GLOBALCONSTANTS Manufacturer_IDs (* ISOBUS Manufacturer ID defines *)
  (* Standard: 61499-1 *)
  (* Version 1.0, 2026-06-29, Franz Höpfinger, Demmler Andreas Fahrzeugbau *)
  PACKAGE isobus::pgn::const;
  VAR_GLOBAL CONSTANT
    M_FOR_EXPERIMENTAL_OR_DEVELOPMENTAL_USE_ONLY : UINT := 0; (* Manufacturer: For experimental or developmental use only. - 2025-11-06 *)
    M_BENDIX_COMMERCIAL_VEHICLE_SYSTEMS : UINT := 1; (* Manufacturer: Bendix Commercial Vehicle Systems LLC (formerly Allied Signal Inc.) | Location: *)
    M_ALLISON_TRANSMISSION : UINT := 2; (* Manufacturer: Allison Transmission, Inc. | Location: Indianapolis, IN USA - 2015-04-28 *)
    M_AMETEK_US_GAUGE_DIVISION : UINT := 3; (* Manufacturer: Ametek, US Gauge Division | Location: Sellersville, PA USA *)
    M_AMETEK_DIXSON : UINT := 4; (* Manufacturer: Ametek-Dixson | Location: Grand Junction, CO USA *)
    M_AMP : UINT := 5; (* Manufacturer: AMP Inc. | Location: Harrisburg, PA USA *)
    M_BERIFORS_ELECTRONICS : UINT := 6; (* Manufacturer: Berifors Electronics AB | Location: Stockholm, Sweden *)
    M_CASE : UINT := 7; (* Manufacturer: Case Corp. | Location: Burr Ridge, IL USA *)
    M_CATERPILLAR : UINT := 8; (* Manufacturer: Caterpillar Inc. | Location: Peoria, IL USA *)
    M_CHRYSLER : UINT := 9; (* Manufacturer: Chrysler Corp. | Location: Auburn Hills, MI USA *)
    M_CUMMINS : UINT := 10; (* Manufacturer: Cummins Inc (formerly Cummins Engine Co) | Location: Columbus, IN USA *)
    M_DEARBORN_GROUP : UINT := 11; (* Manufacturer: Dearborn Group Inc. | Location: Indianapolis, IN & Farmington Hills, MI USA *)
    M_DEERE_AND_COMPANY_PRECISION_FARMING : UINT := 12; (* Manufacturer: Deere & Company, Precision Farming | Location: East Moline, IL USA *)
    M_DELCO_ELECTRONICS : UINT := 13; (* Manufacturer: Delco Electronics | Location: Kokomo, IN USA *)
    M_DETROIT_DIESEL : UINT := 14; (* Manufacturer: Detroit Diesel Corporation | Location: Detroit, MI USA *)
    M_DICKEY_JOHN : UINT := 15; (* Manufacturer: DICKEY-john Corporation | Location: Auburn, IL USA - 2015-07-27 *)
    M_EATON : UINT := 16; (* Manufacturer: Eaton Corp | Location: Southfield, MI USA *)
    M_EATON_RES_AND_DEV : UINT := 17; (* Manufacturer: Eaton Corp, Corp Res & Dev | Location: Milwaukee, WI USA *)
    M_EATON_TRANSMISSION_DIV : UINT := 18; (* Manufacturer: Eaton Corp, Transmission Div. | Location: Kalamazoo, MI USA *)
    M_EATON_TRUCKING_INFO_SERVICES : UINT := 19; (* Manufacturer: Eaton Corp. Trucking Info Services | Location: Clemmons, NC USA *)
    M_EATON_20 : UINT := 20; (* Manufacturer: Eaton Ltd | Location: Worsley, England *)
    M_ECHLIN_MIDLAND_BRAKE : UINT := 21; (* Manufacturer: Echlin Inc., Midland Brake Inc. | Location: Kansas City, MO USA *)
    M_FORD_MOTOR_ELECTRONIC_CONCEPTS_AND_SYSTEMS : UINT := 22; (* Manufacturer: Ford Motor Co., Electronic Concepts & Systems | Location: Dearborn, MI USA *)
    M_FORD_MOTOR_HEAVY_TRUCK : UINT := 23; (* Manufacturer: Ford Motor Co., Heavy Truck | Location: Dearborn, MI USA *)
    M_FORD_MOTOR_VEHICLE_CONTROLS : UINT := 24; (* Manufacturer: Ford Motor Co., Vehicle Controls | Location: Dearborn, MI USA *)
    M_DAIMLER_TRUCKS_NORTH_AMERICA : UINT := 25; (* Manufacturer: Daimler Trucks North America LLC (formerly Freightliner LLC) | Location: Portland, *)
    M_GENERAL_MOTORS_SERVICE_TECHNOLOGY_GRP : UINT := 26; (* Manufacturer: General Motors Corp, Service Technology Grp | Location: Romulus, MI USA *)
    M_GMC : UINT := 27; (* Manufacturer: GMC | Location: Troy, MI USA *)
    M_GROTE_IND : UINT := 28; (* Manufacturer: Grote Ind. Inc. | Location: Madison, IN USA *)
    M_HINO_MOTORS : UINT := 29; (* Manufacturer: Hino Motors Ltd. | Location: Tokyo, Japan *)
    M_ISUZU_MOTORS : UINT := 30; (* Manufacturer: Isuzu Motors Ltd | Location: Kawasaki, Japan *)
    M_J_POLLAK : UINT := 31; (* Manufacturer: J Pollak Corp | Location: Boston, MA USA *)
    M_JACOBS_VEHICLE_SYSTEMS : UINT := 32; (* Manufacturer: Jacobs Vehicle Systems | Location: Bloomfield, CT USA - 1998-07-01 *)
    M_JOHN_DEERE : UINT := 33; (* Manufacturer: John Deere | Location: Moline, IL USA - 2015-06-29 *)
    M_KELSEY_HAYES : UINT := 34; (* Manufacturer: Kelsey Hayes Co. | Location: Livonia, MI USA *)
    M_KENWORTH_TRUCK : UINT := 35; (* Manufacturer: Kenworth Truck Co. | Location: Kirkland, WA USA *)
    M_LUCAS_IND : UINT := 36; (* Manufacturer: Lucas Ind. | Location: Solihull, W Midlands UK *)
    M_MACK_TRUCKS : UINT := 37; (* Manufacturer: Mack Trucks Inc. | Location: Hagerstown, MD USA *)
    M_MICRO_PROCESSOR_SYSTEMS : UINT := 38; (* Manufacturer: Micro Processor Systems Inc. | Location: Sterling Hts, MI USA *)
    M_MICROFIRM : UINT := 39; (* Manufacturer: Microfirm Inc. | Location: Stillwater, OK USA *)
    M_MOTOROLA_AIEG : UINT := 40; (* Manufacturer: Motorola AIEG Inc. | Location: Northbrook, IL USA *)
    M_MOTOROLA : UINT := 41; (* Manufacturer: Motorola Inc. | Location: Schaumburg, IL USA *)
    M_INTERNATIONAL_TRUCK_AND_ENGINE_ENGINE_ELECTRONICS : UINT := 42; (* Manufacturer: International Truck and Engine Corporation - Engine Electronics (formerly Navistar *)
    M_INTERNATIONAL_TRUCK_AND_ENGINE_VEHICLE_ELECTRONICS : UINT := 43; (* Manufacturer: International Truck and Engine Corporation - Vehicle Electronics (formerly Navistar *)
    M_NIPPONDENSO : UINT := 44; (* Manufacturer: Nippondenso Co. Ltd. | Location: Kariya, Aichi Japan *)
    M_PACCAR : UINT := 45; (* Manufacturer: PACCAR | Location: Mount Vernon, WA USA *)
    M_NOREGON_SYSTEMS : UINT := 46; (* Manufacturer: Noregon Systems, LLC (formerly Noregon Systems, Inc) | Location: Greensboro, NC USA *)
    M_PHILLIPS_SEMICONDUCTOR : UINT := 47; (* Manufacturer: Phillips Semiconductor | Location: Sunnyvale, CA USA *)
    M_POLLAK_ALPHABET : UINT := 48; (* Manufacturer: Pollak Alphabet | Location: El Paso, TX USA *)
    M_RE_AMERICA : UINT := 49; (* Manufacturer: RE America Inc. | Location: Cleveland, OH USA *)
    M_ROBERT_BOSCH : UINT := 50; (* Manufacturer: Robert Bosch Corp | Location: Broadview, IL USA *)
    M_ROBERT_BOSCH_51 : UINT := 51; (* Manufacturer: Robert Bosch GmbH | Location: Stuttgart, Germany *)
    M_MERITOR_AUTOMOTIVE : UINT := 52; (* Manufacturer: Meritor Automotive, Inc. (formerly Rockwell Automotive) | Location: Troy, MI USA - *)
    M_CONTINENTAL_AUTOMOTIVE_SYSTEMS_US : UINT := 53; (* Manufacturer: Continental Automotive Systems US, Inc. (formerly Rockwell Land Transportation) | *)
    M_MERITOR_WABCO : UINT := 54; (* Manufacturer: Meritor Wabco | Location: Troy, MI USA *)
    M_RYDER_SYSTEM : UINT := 55; (* Manufacturer: Ryder System Inc. | Location: Miami, FL USA *)
    M_SAIC : UINT := 56; (* Manufacturer: SAIC | Location: San Diego, CA USA *)
    M_DANFOSS : UINT := 57; (* Manufacturer: Danfoss (formerly Sauer Sundstrand Co, then Sauer-Danfoss Co) | Location: Nordborg, *)
    M_SPX_OTC_DIV : UINT := 58; (* Manufacturer: SPX Corporation, OTC Div | Location: Owatonna, MN USA *)
    M_VES : UINT := 59; (* Manufacturer: VES Inc. | Location: Rock Hill, SC USA *)
    M_VOLVO_TRUCKS_NORTH_AMERICA : UINT := 60; (* Manufacturer: Volvo Trucks North America Inc. | Location: Greensboro, NC USA - 1999-02-01 *)
    M_VOLVO_TRUCK : UINT := 61; (* Manufacturer: Volvo Truck Corp. | Location: Gothenburg, Sweden *)
    M_WABCO : UINT := 62; (* Manufacturer: Wabco | Location: Hanover, Germany *)
    M_ZF_INDUSTRIES : UINT := 63; (* Manufacturer: ZF Industries Inc. | Location: Vernon Hills, IL USA *)
    M_UNUSED_64 : UINT := 64; (* Manufacturer: Unused (formerly SpectraPrecision Laserplane, then SpectraPhysics) - 2001-02-15 *)
    M_MAN_NUTZFAHRZEUGE_AG : UINT := 65; (* Manufacturer: MAN Nutzfahrzeuge AG | Location: Munich, Germany - 1999-02-01 *)
    M_JOHN_DEERE_CONSTRUCTION_EQUIPMENT_DIVISION : UINT := 66; (* Manufacturer: John Deere Construction Equipment Division | Location: Dubuque, IA USA - 1999-11-11 *)
    M_JOHN_DEERE_COFFEYVILLE_WORKS : UINT := 67; (* Manufacturer: John Deere Coffeyville Works (formerly Funk Manufacturing Company) | Location: *)
    M_SCANIA : UINT := 68; (* Manufacturer: Scania | Location: Södertälje, Sweden *)
    M_TRIMBLE_NAVIGATION : UINT := 69; (* Manufacturer: Trimble Navigation *)
    M_FLEX_COIL_LIMITED : UINT := 70; (* Manufacturer: Flex-coil Limited | Location: Saskatoon, SK Canada *)
    M_VANSCO_ELECTRONICS : UINT := 71; (* Manufacturer: Vansco Electronics Ltd. | Location: Winnipeg, MB Canada *)
    M_SISU : UINT := 72; (* Manufacturer: Sisu Corporation | Location: ESPOO, Finland *)
    M_LETOURNEAU : UINT := 73; (* Manufacturer: LeTourneau, Inc. | Location: Longview, TX USA *)
    M_EATON_AXLE_BRAKE_DIVISION : UINT := 74; (* Manufacturer: Eaton Axle-Brake Division | Location: Kalamazoo, MI USA *)
    M_DEERE_AND_AGRICULTURAL_DIVISION : UINT := 75; (* Manufacturer: Deere & Co, Agricultural Division - 1998-02-01 *)
    M_UNUSED_76 : UINT := 76; (* Manufacturer: unused (formerly Deere & Co, Construction Division) - 1999-11-11 *)
    M_DEERE_POWER_SYSTEMS_GROUP : UINT := 77; (* Manufacturer: Deere Power Systems Group - 1998-02-01 *)
    M_FRANK_W_MURPHY_MANUFACTURING : UINT := 78; (* Manufacturer: Frank W. Murphy Manufacturing, Inc | Location: Tulsa, OK USA - 1998-02-01 *)
    M_DAIMLER_BENZ_AG_ENGINE_DIVISION : UINT := 79; (* Manufacturer: Daimler Benz AG - Engine Division (PBM) | Location: Stuttgart, Germany - 1998-02-01 *)
    M_TWIN_DISC : UINT := 80; (* Manufacturer: Twin Disc, Inc. | Location: Racine, WI USA - 1998-04-01 *)
    M_FIRE_RESEARCH : UINT := 81; (* Manufacturer: Fire Research Corp. | Location: Nesconset, NY USA - 1998-04-01 *)
    M_BOBCAT_INGERSOLL_RAND : UINT := 82; (* Manufacturer: Bobcat/Ingersoll-Rand (formerly Melroe/Ingersoll-Rand) | Location: Fargo, ND USA - *)
    M_BENDIX_VORAD_TECHNOLOGIES : UINT := 83; (* Manufacturer: Bendix VORAD Technologies (formerly Eaton VORAD Technologies) | Location: San *)
    M_NEW_HOLLAND_UK_LIMITED : UINT := 84; (* Manufacturer: New Holland UK Limited | Location: Basildon, Essex UK - 1999-11-11 *)
    M_KOHLER : UINT := 85; (* Manufacturer: Kohler Co | Location: Kohler, WI USA - 1999-11-11 *)
    M_C_E_NIEHOFF_AND_COMPANY : UINT := 86; (* Manufacturer: C. E. Niehoff & Company | Location: Evanston, IL USA - 1999-11-11 *)
    M_J_C_BAMFORD_EXCAVATORS : UINT := 87; (* Manufacturer: J.C. Bamford Excavators Ltd (JCB) | Location: Rocester, Staffordshire UK - *)
    M_HEMISPHERE_GPS : UINT := 88; (* Manufacturer: Hemisphere GPS Inc (formerly Satloc Precision GPS) | Location: Scottsdale, AZ USA - *)
    M_KVERNELAND_GROUP_ELECTRONICS_DIVISION : UINT := 89; (* Manufacturer: Kverneland Group, Electronics Division | Location: Nieuw-Vennep, The Netherlands - *)
    M_KNORR_BREMSE_SFN : UINT := 90; (* Manufacturer: Knorr-Bremse SfN GmbH | Location: Munich, Germany - 2000-05-11 *)
    M_BSG_BODENSEE_STEUERGERAETE : UINT := 91; (* Manufacturer: BSG Bodensee Steuergeraete GmbH | Location: Immenstaad, Germany - 2000-05-11 *)
    M_AG_CHEM_EQUIPMENT : UINT := 92; (* Manufacturer: Ag-Chem Equipment Co., Inc. | Location: Duluth, GA USA - 2015-08-20 *)
    M_PERKINS_ENGINES_COMPANY : UINT := 93; (* Manufacturer: Perkins Engines Company Ltd. | Location: Peterborough, UK - 2000-08-10 *)
    M_CNH_INDUSTRIAL_N_V : UINT := 94; (* Manufacturer: CNH Industrial N.V. (formerly CNH Global N.V.) | Location: Racine, WI USA - *)
    M_PACIFIC_INSIGHT_ELECTRONICS : UINT := 95; (* Manufacturer: Pacific Insight Electronics Corp. | Location: Nelson, BC Canada - 2000-08-10 *)
    M_MECH_TRONIC_IT : UINT := 96; (* Manufacturer: Mech@tronic IT GmbH | Location: Hetzenhausen, Germany - 2000-11-09 *)
    M_AG_LEADER_TECHNOLOGY : UINT := 97; (* Manufacturer: Ag Leader Technology, Inc. | Location: Ames, IA USA - 2000-11-09 *)
    M_PTX_TRIMBLE : UINT := 98; (* Manufacturer: PTx Trimble (formerly Mueller-Elektronik GmbH & Co) | Location: Westminster, CO USA *)
    M_INTERNATIONAL_TRANSMISSIONS : UINT := 99; (* Manufacturer: International Transmissions Ltd (ITL) | Location: Wrexham, North Wales UK - *)
    M_VDO_TECHNIK_AG : UINT := 100; (* Manufacturer: VDO Technik AG | Location: Rüthi, Switzerland - 2001-02-21 *)
    M_SENSORIA : UINT := 101; (* Manufacturer: Sensoria | Location: San Diego, CA USA - 2001-02-21 *)
    M_AGCO : UINT := 102; (* Manufacturer: AGCO (formerly AGCO GmbH & Co.) | Location: Duluth, GA USA - 2015-08-20 *)
    M_CLAAS_E_SYSTEMS : UINT := 103; (* Manufacturer: CLAAS E-Systems GmbH (formerly CLAAS E-Systems KGaA mbH & Co. KG) | Location: *)
    M_CLAAS_KGAA_MBH : UINT := 104; (* Manufacturer: CLAAS KGaA mbH (formerly CLAAS Selbstfahrende Erntemaschinen GmbH) | Location: *)
    M_KIEPE_ELEKTRIK_AND : UINT := 105; (* Manufacturer: Kiepe Elektrik GmbH & Co. KG | Location: Duesseldorf, Germany - 2001-05-25 *)
    M_BAE_SYSTEMS_CONTROLS : UINT := 106; (* Manufacturer: BAE Systems Controls, Inc. | Location: Endicott, NY USA - 2015-06-12 *)
    M_GRIMME_LANDMASCHINEN_AND : UINT := 107; (* Manufacturer: Grimme Landmaschinen GmbH & Co. KG | Location: Damme, Germany - 2001-06-28 *)
    M_PTX_TRIMBLE_108 : UINT := 108; (* Manufacturer: PTx Trimble (formerly WTK-Elecktronik GmbH, now a duplicate entry; use MFR ID 98) | *)
    M_TEEJET_TECHNOLOGIES_DENMARK : UINT := 109; (* Manufacturer: TeeJet Technologies Denmark (formerly LH Technologies ApS) | Location: Aabybro, *)
    M_EPIQ_SENSOR_NITE : UINT := 110; (* Manufacturer: EPIQ Sensor-Nite | Location: Fenton, MI USA - 2001-09-19 *)
    M_BERNARD_KRONE_HOLDING_SE_AND : UINT := 111; (* Manufacturer: Bernard Krone Holding SE & Co. KG (formerly Maschinenfabrik Bernard Krone GmbH) | *)
    M_MECALAC : UINT := 112; (* Manufacturer: MECALAC | Location: Annecy le Vieux, France - 2001-12-31 *)
    M_STRESS_TEK : UINT := 113; (* Manufacturer: Stress-Tek, Inc. | Location: Kent, WA USA - 2002-01-14 *)
    M_ECONTROLS : UINT := 114; (* Manufacturer: EControls, Inc. | Location: San Antonio, TX USA - 2002-04-21 *)
    M_NACCO_MATERIALS_HANDLING_GROUP : UINT := 115; (* Manufacturer: NACCO Materials Handling Group, Inc. | Location: Portland, OR USA - 2002-05-01 *)
    M_BEELINE_TECHNOLOGIES : UINT := 116; (* Manufacturer: BEELINE Technologies | Location: Brisbane, QLD Australia - 2002-05-01 *)
    M_HUSCO_INTERNATIONAL : UINT := 117; (* Manufacturer: HUSCO International | Location: Waukesha, WI USA - 2002-05-29 *)
    M_INTRON : UINT := 118; (* Manufacturer: Intron GmbH | Location: Schwaebisch Hall, Germany - 2002-07-28 *)
    M_INTEGRINAUTICS : UINT := 119; (* Manufacturer: IntegriNautics | Location: Menlo Park, CA USA - 2002-07-30 *)
    M_RDS_TECHNOLOGY : UINT := 120; (* Manufacturer: RDS Technology Ltd | Location: Minchinhampton, Stroud UK - 2002-08-24 *)
    M_HED : UINT := 121; (* Manufacturer: HED (Hydro Electronic Devices, Inc.) | Location: Hartford, WI USA - 2002-09-02 *)
    M_FG_WILSON_LIMITED : UINT := 122; (* Manufacturer: FG Wilson (Engineering) Limited | Location: Larne, County Antrim UK - 2002-09-13 *)
    M_BASLER_ELECTRIC : UINT := 123; (* Manufacturer: Basler Electric | Location: Highland, IL USA - 2002-11-09 *)
    M_HYDAC_ELECTRONIC : UINT := 124; (* Manufacturer: Hydac Electronic | Location: Saarbruecken, Germany - 2003-01-28 *)
    M_NEVADA_AUTOMOTIVE_TEST_CENTER : UINT := 125; (* Manufacturer: Nevada Automotive Test Center | Location: Carson City, NV USA - 2003-02-20 *)
    M_DRIVER_TECH : UINT := 126; (* Manufacturer: Driver Tech | Location: Salt Lake City, UT USA - 2003-02-20 *)
    M_HOLLAND_USA : UINT := 127; (* Manufacturer: Holland USA | Location: Holland, MI USA - 2003-03-29 *)
    M_GERHARD_DUECKER_AND : UINT := 128; (* Manufacturer: Gerhard Duecker GmbH & Co. KG | Location: Stadtlohn, Germany - 2003-03-29 *)
    M_OMNEX_CONTROL_SYSTEMS : UINT := 129; (* Manufacturer: OMNEX Control Systems Inc. | Location: Port Coquitlam, BC Canada - 2003-03-31 *)
    M_NIDO_UNIVERSAL_MACHINES_B_V : UINT := 130; (* Manufacturer: Nido - Universal Machines B.V. | Location: Holten, The Netherlands - 2003-04-28 *)
    M_ITT_INDUSTRIES : UINT := 131; (* Manufacturer: ITT Industries | Location: Eden Prarie, MN USA - 2003-06-05 *)
    M_MULAG_FAHRZEUGWERK : UINT := 132; (* Manufacturer: Mulag-Fahrzeugwerk | Location: Oppenau, Germany - 2003-07-13 *)
    M_BUCHER_SCHOERLING : UINT := 133; (* Manufacturer: Bucher Schoerling GmbH | Location: Hannover, Germany - 2003-07-13 *)
    M_IRIS_TECHNOLOGY : UINT := 134; (* Manufacturer: Iris Technology Ltd | Location: Lancaster, Lancs UK - 2003-07-20 *)
    M_AIRMAR_TECHNOLOGY : UINT := 135; (* Manufacturer: Airmar Technology Corporation | Location: Milford, NH USA - 2003-08-20 *)
    M_KOMATSU : UINT := 136; (* Manufacturer: Komatsu Ltd | Location: Hiratsuka, Kanagawa Japan - 2003-08-20 *)
    M_MARETRON : UINT := 137; (* Manufacturer: Maretron | Location: Phoenix AZ USA *)
    M_GEORG_FRITZMEIER_AND : UINT := 138; (* Manufacturer: Georg Fritzmeier GmbH & Co. KG | Location: Grosshelfendorf, Germany - 2003-09-15 *)
    M_CATERPILLAR_TRIMBLE_CONTROL_TECHNOLOGIES : UINT := 139; (* Manufacturer: Caterpillar Trimble Control Technologies (CTCT), LLC | Location: Dayton, OH USA - *)
    M_LOWRANCE_ELECTRONICS : UINT := 140; (* Manufacturer: Lowrance Electronics, Inc. | Location: Tulsa, OK USA - 2003-09-18 *)
    M_THALES_NAVIGATION : UINT := 141; (* Manufacturer: Thales Navigation Ltd. | Location: Surrey, UK - 2003-11-01 *)
    M_TRW_AUTOMOTIVE : UINT := 142; (* Manufacturer: TRW Automotive (Commercial Steering Systems) | Location: Lafayette, IN USA - *)
    M_W_GMEINER_AND : UINT := 143; (* Manufacturer: W. Gmeiner GmbH & Co. | Location: Kummersbruck, Germany - 2003-12-20 *)
    M_MERCURY_MARINE : UINT := 144; (* Manufacturer: Mercury Marine | Location: Fond du Lac, WI USA - 2003-12-20 *)
    M_MURCAL_CONTROLS : UINT := 145; (* Manufacturer: MurCal Controls | Location: Palmdale, CA USA - 2003-12-31 *)
    M_MAXIMA_TECHNOLOGIES : UINT := 146; (* Manufacturer: Maxima Technologies | Location: Lancaster, PA USA - 2004-01-12 *)
    M_NAUTIBUS_ELECTRONIC : UINT := 147; (* Manufacturer: Nautibus electronic GmbH | Location: Quern, Germany - 2004-01-24 *)
    M_BLUE_WATER_DATA : UINT := 148; (* Manufacturer: Blue Water Data, Inc. | Location: Salem, NJ USA - 2004-01-24 *)
    M_HOLSET : UINT := 149; (* Manufacturer: Holset | Location: Charleston, SC USA - 2004-01-24 *)
    M_FLEETGUARD : UINT := 150; (* Manufacturer: Fleetguard | Location: Nashville, TN USA - 2004-01-24 *)
    M_RAVEN_INDUSTRIES : UINT := 151; (* Manufacturer: Raven Industries, Inc. | Location: Sioux Falls, SD USA - 2015-09-08 *)
    M_ELOBAU_AND : UINT := 152; (* Manufacturer: elobau GmbH & Co. KG | Location: Leutkirch, Germany - 2009-11-30 *)
    M_WOODWARD_INDUSTRIAL_CONTROLS_DIVISION : UINT := 153; (* Manufacturer: Woodward, Industrial Controls Division | Location: Fort Collins, CO USA - *)
    M_WESTERBEKE : UINT := 154; (* Manufacturer: Westerbeke Corporation | Location: Taunton, MA USA - 2004-05-01 *)
    M_VETRONIX : UINT := 155; (* Manufacturer: Vetronix Corporation | Location: Santa Barbara, CA - 2004-05-24 *)
    M_ITT_INDUSTRIES_CANNON : UINT := 156; (* Manufacturer: ITT Industries - Cannon | Location: Shakopee, MN USA - 2004-07-20 *)
    M_ISSPRO : UINT := 157; (* Manufacturer: ISSPRO Inc. | Location: Portland, OR USA - 2004-07-20 *)
    M_FIRESTONE_INDUSTRIAL_PRODUCTS_COMPANY : UINT := 158; (* Manufacturer: Firestone Industrial Products Company | Location: Carmel, IN USA - 2004-10-05 *)
    M_NTECH_INDUSTRIES : UINT := 159; (* Manufacturer: NTech Industries Inc | Location: Ukiah, CA USA - 2004-10-05 *)
    M_NIDO : UINT := 160; (* Manufacturer: Nido | Location: Holten, The Netherlands - 2004-10-05 *)
    M_OFFSHORE_SYSTEMS : UINT := 161; (* Manufacturer: Offshore Systems (UK) Ltd | Location: New Milton, Hampshire UK - 2004-10-05 *)
    M_AXIOMATIC_TECHNOLOGIES : UINT := 162; (* Manufacturer: Axiomatic Technologies | Location: Mississauga, ON Canada - 2004-10-05 *)
    M_BRP : UINT := 163; (* Manufacturer: BRP Inc. | Location: Waukegan, IL USA - 2004-10-05 *)
    M_MTU_FRIEDRICHSHAFEN : UINT := 164; (* Manufacturer: MTU Friedrichshafen GmbH (formerly DaimlerChrysler Off-Highway) | Location: *)
    M_CPAC_SYSTEMS : UINT := 165; (* Manufacturer: CPAC Systems AB | Location: Vastra Frolunda, Sweden - 2004-10-05 *)
    M_JOHN_DEERE_ELECTRONIC_SOLUTIONS : UINT := 166; (* Manufacturer: John Deere Electronic Solutions (formerly Phoenix International) | Location: Fargo, *)
    M_JLG_INDUSTRIES : UINT := 167; (* Manufacturer: JLG Industries Inc | Location: McConnellsburg, PA USA - 2004-10-20 *)
    M_XANTREX : UINT := 168; (* Manufacturer: Xantrex | Location: Burnaby, BC Canada - 2004-12-15 *)
    M_MARLIN_TECHNOLOGIES : UINT := 169; (* Manufacturer: Marlin Technologies Inc. | Location: Horicon, WI USA - 2004-12-15 *)
    M_COMPUTRONICS : UINT := 170; (* Manufacturer: Computronics Corporation Ltd. | Location: Bentley, WA Australia - 2004-12-15 *)
    M_TOPCON_ELECTRONICS_AND : UINT := 171; (* Manufacturer: Topcon Electronics GmbH & Co. KG (formerly Wachendorff Elektronik GmbH & Co. KG) | *)
    M_YANMAR : UINT := 172; (* Manufacturer: Yanmar Co., Ltd. (formerly Yanmar Marine USA) | Location: Maibara, Shiga Japan - *)
    M_RYESO : UINT := 173; (* Manufacturer: Ryeso, Inc. | Location: Palmdale, CA USA - 2005-01-20 *)
    M_VOLVO_PENTA : UINT := 174; (* Manufacturer: AB Volvo Penta | Location: Goteburg, Sweden - 2005-01-20 *)
    M_VERIS_TECHNOLOGIES : UINT := 175; (* Manufacturer: Veris Technologies, Inc. | Location: Salina, KS USA - 2005-01-20 *)
    M_MORITZ_AEROSPACE : UINT := 176; (* Manufacturer: Moritz Aerospace | Location: Dublin, PA USA - 2005-01-25 *)
    M_DIAGNOSTIC_SYSTEMS_ASSOCIATES : UINT := 177; (* Manufacturer: Diagnostic Systems Associates | Location: Kalamazoo, MI USA - 2005-03-02 *)
    M_CONTINENTAL_AUTOMOTIVE : UINT := 178; (* Manufacturer: Continental Automotive GmbH (formerly Siemens VDO Automotive AG) | Location: *)
    M_TEEJET_TECHNOLOGIES_SPRINGFIELD : UINT := 179; (* Manufacturer: TeeJet Technologies Springfield (formerly Midwest Technologies Illinois, LLC) | *)
    M_SMART_POWER_SYSTEMS : UINT := 180; (* Manufacturer: Smart Power Systems | Location: Reed City, MI USA - 2005-04-15 *)
    M_CORETRONICS : UINT := 181; (* Manufacturer: Coretronics, Inc. | Location: Eagle, ID USA - 2005-04-15 *)
    M_VEHICLE_SYSTEMS_ENGINEERING_B_V : UINT := 182; (* Manufacturer: Vehicle Systems Engineering B.V. | Location: Veenendaal, The Netherlands - *)
    M_KDS_CONTROLS : UINT := 183; (* Manufacturer: KDS Controls, Inc | Location: Troy, MI USA - 2005-06-05 *)
    M_EIA_ELECTRONICS : UINT := 184; (* Manufacturer: EIA Electronics | Location: Aartselaar, Belguim - 2005-06-21 *)
    M_BEEDE_ELECTRICAL_INSTRUMENT_COMPANY : UINT := 185; (* Manufacturer: Beede Electrical Instrument Company | Location: Penacock, NH USA - 2005-07-01 *)
    M_ALTRONIC : UINT := 186; (* Manufacturer: Altronic, Inc | Location: Girard, OH USA - 2005-08-01 *)
    M_AIR_WEIGH : UINT := 187; (* Manufacturer: Air-Weigh | Location: Eugene, OR USA - 2005-08-12 *)
    M_EMP : UINT := 188; (* Manufacturer: EMP Corp | Location: Escanaba, MI USA - 2005-08-12 *)
    M_QUALCOMM : UINT := 189; (* Manufacturer: QUALCOMM | Location: San Diego, CA USA - 2005-08-12 *)
    M_HELLA_KGAA_HUECK_AND : UINT := 190; (* Manufacturer: Hella KGaA Hueck & Co | Location: Lippstadt, Germany - 2005-08-12 *)
    M_XRS : UINT := 191; (* Manufacturer: XRS Corporation (formerly XATA Corporation) | Location: Eden Prairie, MN USA - *)
    M_FLOSCAN : UINT := 192; (* Manufacturer: Floscan | Location: Seattle, WA USA - 2005-08-31 *)
    M_JEPPESEN_MARINE : UINT := 193; (* Manufacturer: Jeppesen Marine | Location: Portland, OR USA - 2005-08-31 *)
    M_TRIMARK : UINT := 194; (* Manufacturer: TriMark Corporation | Location: New Hampton, IA USA - 2005-08-31 *)
    M_GENERAL_ENGINE_PRODUCTS : UINT := 195; (* Manufacturer: General Engine Products | Location: Livonia, MI USA - 2005-10-21 *)
    M_LEMKEN_AND : UINT := 196; (* Manufacturer: LEMKEN GmbH & Co KG | Location: Alpen, Germany - 2005-10-21 *)
    M_MECHRON_POWER_SYSTEMS : UINT := 197; (* Manufacturer: Mechron Power Systems | Location: Ottawa, ON Canada - 2005-10-21 *)
    M_MYSTIC_VALLEY_COMMUNICATIONS : UINT := 198; (* Manufacturer: Mystic Valley Communications | Location: Mystic, CT USA - 2005-10-21 *)
    M_ACTIA_GROUP : UINT := 199; (* Manufacturer: ACTIA Group (formerly Actia Corp) | Location: Toulouse, France - 2017-07-11 *)
    M_MGM_BRAKES : UINT := 200; (* Manufacturer: MGM Brakes | Location: Charlotte, NC USA - 2005-11-01 *)
    M_DISENOS_Y_TECNOLOGIA : UINT := 201; (* Manufacturer: Disenos y Tecnologia S.A. | Location: Barcelona, Spain - 2005-11-10 *)
    M_CURTIS_INSTRUMENTS : UINT := 202; (* Manufacturer: Curtis Instruments, Inc | Location: Mount Kisco, NY USA - 2005-11-14 *)
    M_MILTRONIK : UINT := 203; (* Manufacturer: MILtronik GmbH | Location: Hilden, Germany - 2006-01-03 *)
    M_THE_MOREY : UINT := 204; (* Manufacturer: The Morey Corporation | Location: Woodridge, IL USA - 2006-01-13 *)
    M_SMARTIRE_SYSTEMS : UINT := 205; (* Manufacturer: SmarTire Systems Inc | Location: Richmond, BC Canada - 2006-01-13 *)
    M_PORT : UINT := 206; (* Manufacturer: port GmbH | Location: Halle, Germany - 2006-02-02 *)
    M_OTTO_ENGINEERING : UINT := 207; (* Manufacturer: Otto Engineering | Location: Carpentersville, IL USA - 2006-02-09 *)
    M_DREW_TECHNOLOGIES : UINT := 208; (* Manufacturer: Drew Technologies, Inc | Location: Whitmore Lake, MI USA - 2006-02-09 *)
    M_BELL_EQUIP : UINT := 209; (* Manufacturer: Bell Equip. Co. SA (PTY) LTD | Location: Richards Bay, South Africa - 2006-03-14 *)
    M_ITERIS : UINT := 210; (* Manufacturer: Iteris, Inc. | Location: Anaheim, CA USA - 2006-03-14 *)
    M_DNA_GROUP : UINT := 211; (* Manufacturer: DNA Group | Location: Raleigh, NC USA - 2006-03-22 *)
    M_SURE_POWER_INDUSTRIES : UINT := 212; (* Manufacturer: Sure Power Industries, Inc | Location: Tualatin, OR USA - 2006-03-22 *)
    M_CNH_BELGIUM_N_V : UINT := 213; (* Manufacturer: CNH Belgium N.V. | Location: Zedelgem, Belgium - 2006-03-24 *)
    M_MC_ELETTRONICA_SRL : UINT := 214; (* Manufacturer: MC elettronica Srl | Location: Fiesso Umbertiano, Rovigo, Italy - 2006-03-24 *)
    M_AETNA_ENGINEERING_FIREBOY_XINTEX : UINT := 215; (* Manufacturer: Aetna Engineering/Fireboy-Xintex | Location: Grand Rapids, MI USA - 2006-04-03 *)
    M_PANELTRONICS : UINT := 216; (* Manufacturer: Paneltronics Inc. | Location: Hialeah Gardens, FL USA - 2006-04-02 *)
    M_RM_MICHAELIDES_SOFTWARE_AND_ELEKTRONIK : UINT := 217; (* Manufacturer: RM Michaelides Software & Elektronik GmbH | Location: Fulda, Germany - 2006-04-21 *)
    M_GITS_MANUFACTURING_COMPANY : UINT := 218; (* Manufacturer: Gits Manufacturing Company | Location: Creston, IA USA - 2006-04-21 *)
    M_CAT_OEM_SOLUTIONS : UINT := 219; (* Manufacturer: Cat OEM Solutions | Location: Mossville, IL USA - 2006-04-25 *)
    M_BEEDE_ELECTRICAL_INSTRUMENT_COMPANY_220 : UINT := 220; (* Manufacturer: Beede Electrical Instrument Company, Inc | Location: Penacook, NH USA - 2006-04-29 *)
    M_SIE : UINT := 221; (* Manufacturer: SiE | Location: Kempten/Allgaeu, Germany - 2006-06-05 *)
    M_GENERAC_POWER_SYSTEMS : UINT := 222; (* Manufacturer: Generac Power Systems, Inc. | Location: Waukesha, WI, USA - 2006-08-03 *)
    M_VAUEO_RETARDER : UINT := 223; (* Manufacturer: Vaueo Retarder Co., Ltd. | Location: Shajin, Baoan, Shen Zhen China - 2006-08-20 *)
    M_EMMI_NETWORK_S_L : UINT := 224; (* Manufacturer: EMMI Network, S.L. | Location: Gandia, Spain - 2006-08-20 *)
    M_SKF : UINT := 225; (* Manufacturer: SKF | Location: Gothenburg, Sweden - 2006-08-31 *)
    M_MONACO_COACH : UINT := 226; (* Manufacturer: Monaco Coach Corporation | Location: Bend, OR USA - 2006-09-16 *)
    M_LYKKETRONIC : UINT := 227; (* Manufacturer: Lykketronic A/S | Location: Loegstoer, Denmark - 2006-10-15 *)
    M_UNUSED_228 : UINT := 228; (* Manufacturer: Unused (formerly ZF Marine Electronics) - 2015-07-27 *)
    M_GARMIN_INTERNATIONAL : UINT := 229; (* Manufacturer: Garmin International Inc. | Location: Olathe, KS USA - 2006-10-15 *)
    M_SAUCON_TECHNOLOGIES : UINT := 230; (* Manufacturer: Saucon Technologies | Location: Bethlehem, PA USA - 2006-11-06 *)
    M_TOPCON_POSITIONING_SYSTEMS : UINT := 231; (* Manufacturer: Topcon Positioning Systems, Inc. | Location: Livermore, CA USA - 2006-11-13 *)
    M_TSD_INTEGRATED_CONTROLS : UINT := 232; (* Manufacturer: TSD Integrated Controls | Location: Minneapolis, MN USA - 2006-11-13 *)
    M_YACHT_MONITORING_SOLUTIONS : UINT := 233; (* Manufacturer: Yacht Monitoring Solutions Inc. | Location: Corpus Christi, TX USA - 2006-11-14 *)
    M_MONDIAL_ELECTRONIC : UINT := 234; (* Manufacturer: Mondial electronic GmbH | Location: Eggelsberg, Austria - 2006-12-22 *)
    M_SAILORMADE_MARINE_TELEMETRY_TETRA_TECHNOLOGY : UINT := 235; (* Manufacturer: SailorMade Marine Telemetry - Tetra Technology Ltd. | Location: Florianopolis, *)
    M_NORAC_SYSTEMS_INTERNATIONAL : UINT := 236; (* Manufacturer: NORAC Systems International Inc | Location: Saskatoon, SK Canada - 2015-07-27 *)
    M_AGTRON_ENTERPRISES : UINT := 237; (* Manufacturer: Agtron Enterprises Inc | Location: Saskatoon, SK Canada - 2007-01-20 *)
    M_ZF_FRIEDRICHSHAFEN_AG : UINT := 238; (* Manufacturer: ZF Friedrichshafen AG | Location: Friedrichshafen, Germany - 2007-01-20 *)
    M_MAY_AND_SCOFIELD : UINT := 239; (* Manufacturer: May & Scofield Ltd | Location: Basingstoke, Hants, UK - 2007-01-20 *)
    M_VANAIR_MFG : UINT := 240; (* Manufacturer: Vanair Mfg | Location: New Buffalo, MI USA - 2007-01-20 *)
    M_SCHNEIDER_AUTOMATION_SAS : UINT := 241; (* Manufacturer: Schneider Automation SAS | Location: Sophia Antipolis, France - 2007-01-20 *)
    M_KOKUSANDENKI : UINT := 242; (* Manufacturer: Kokusandenki Co. Ltd | Location: Numazu, Shizuoka Japan - 2007-01-20 *)
    M_ERIDE : UINT := 243; (* Manufacturer: eRide, Inc. | Location: San Francisco, CA USA - 2007-02-18 *)
    M_TECHNO_MATIC : UINT := 244; (* Manufacturer: Techno-Matic | Location: Aars, Denmark - 2007-03-11 *)
    M_CAPSTAN_AG_SYSTEMS : UINT := 245; (* Manufacturer: Capstan Ag Systems, Inc. | Location: Topeka, KS USA - 2007-03-11 *)
    M_CLASS_1 : UINT := 246; (* Manufacturer: Class 1, Inc | Location: Ocala, FL USA - 2007-04-24 *)
    M_EPULSE : UINT := 247; (* Manufacturer: ePULSE | Location: Troy, MI USA - 2007-04-29 *)
    M_COOPER_STANDARD_AUTOMOTIVE_ACTIVE_SYSTEMS_GROUP : UINT := 248; (* Manufacturer: Cooper Standard Automotive Active Systems Group | Location: Mitchell, ON Canada - *)
    M_SCHALTBAU : UINT := 249; (* Manufacturer: Schaltbau GmbH | Location: Munich, Germany - 2007-06-15 *)
    M_KUHN_GROUP : UINT := 250; (* Manufacturer: Kuhn Group | Location: Saverne, France - 2007-06-15 *)
    M_GERMAN_AGRICULTURAL_SOCIETY_TEST_CENTER : UINT := 251; (* Manufacturer: German Agricultural Society, Test Center (DLG) | Location: Gross-Ultstadt, Germany *)
    M_SENSOR_TECHNIK_WIEDEMANN : UINT := 252; (* Manufacturer: Sensor-Technik Wiedemann GmbH | Location: Kaufbeuren, Germany - 2007-06-15 *)
    M_MOBILE_CONTROL_SYSTEMS : UINT := 253; (* Manufacturer: Mobile Control Systems | Location: Brussels, Belgium - 2007-06-15 *)
    M_GE_SENSING : UINT := 254; (* Manufacturer: GE Sensing | Location: St. Marys, PA USA - 2007-06-18 *)
    M_MEAS_FRANCE : UINT := 255; (* Manufacturer: MEAS France | Location: Toulouse, France - 2007-07-20 *)
    M_TYCO_ELECTRONICS_AMP : UINT := 256; (* Manufacturer: Tyco Electronics AMP | Location: Osan-Si, Kyunggi-Do, Korea - 2007-07-20 *)
    M_HONDA_MOTOR : UINT := 257; (* Manufacturer: Honda Motor Co., Ltd | Location: Wako-city, Saitama Japan - 2007-07-28 *)
    M_ARAG : UINT := 258; (* Manufacturer: ARAG | Location: Rubiera, Italy - 2007-08-13 *)
    M_BUCHER_AUTOMATION_AG : UINT := 259; (* Manufacturer: Bucher Automation AG (formerly Jetter AG) | Location: Ludwigsburg, Germany - *)
    M_REICHHARDT_STEUERUNGSTECHNIK : UINT := 260; (* Manufacturer: Reichhardt GmbH Steuerungstechnik | Location: Hungen, Germany - 2007-08-13 *)
    M_RED_DOT : UINT := 261; (* Manufacturer: Red Dot Corporation | Location: Seattle, WA USA - 2007-08-13 *)
    M_HYDRAFORCE : UINT := 262; (* Manufacturer: HydraForce, Inc | Location: Lincolnshire, IL USA - 2007-08-13 *)
    M_IMMI : UINT := 263; (* Manufacturer: IMMI | Location: Westfield, IN USA - 2007-08-14 *)
    M_AUTOLYNC : UINT := 264; (* Manufacturer: Autolync | Location: Clayton, Victoria Australia - 2007-09-03 *)
    M_MTS_SENSOR_TECHNOLOGIE : UINT := 265; (* Manufacturer: MTS Sensor Technologie GmbH | Location: Luedenscheid, Germany - 2007-09-05 *)
    M_INTERNATIONAL_THERMAL_RESEARCH : UINT := 266; (* Manufacturer: International Thermal Research Ltd | Location: Richmond, BC Canada - 2007-09-27 *)
    M_RED_LION_CONTROLS : UINT := 267; (* Manufacturer: Red Lion Controls, Inc | Location: York, PA USA - 2007-09-27 *)
    M_ACCURATE_TECHNOLOGIES : UINT := 268; (* Manufacturer: Accurate Technologies | Location: Wixom, MI USA - 2007-10-13 *)
    M_SAFT_AMERICA_SPACE_AND_DEFENSE_DIVISION : UINT := 269; (* Manufacturer: Saft America Inc., Space & Defense Division | Location: Cockeysville, MD USA - *)
    M_TENNANT : UINT := 270; (* Manufacturer: Tennant | Location: Minneapolis, MN USA - 2007-11-10 *)
    M_COLE_HERSEE : UINT := 271; (* Manufacturer: Cole Hersee | Location: South Boston, MA USA - 2007-11-10 *)
    M_GROSS_MECHANICAL_LABORATORIES : UINT := 272; (* Manufacturer: Gross Mechanical Laboratories, Inc | Location: Hanover, MD USA - 2007-11-30 *)
    M_ACTIVE_RESEARCH_LIMITED : UINT := 273; (* Manufacturer: Active Research Limited | Location: Poole, Dorset, UK - 2007-11-30 *)
    M_LTW_TECHNOLOGY : UINT := 274; (* Manufacturer: LTW Technology Co., LTD | Location: Shinjuang City, Taipei Hsien, Taiwan R.O.C. - *)
    M_NAVICO_EGERSUND : UINT := 275; (* Manufacturer: Navico Egersund AS | Location: Egersund, Norway - 2007-12-17 *)
    M_AQUA_HOT_HEATING_SYSTEMS : UINT := 276; (* Manufacturer: Aqua-Hot Heating Systems | Location: Fort Lupton, CO USA - 2008-01-27 *)
    M_LHP_TELEMATICS : UINT := 277; (* Manufacturer: LHP Telematics | Location: Columbus, IN USA - 2008-01-27 *)
    M_TAKATA_ELECTRONICS : UINT := 278; (* Manufacturer: Takata Electronics | Location: Farmington Hills, MI USA - 2008-02-15 *)
    M_GEOMETRIS_LP : UINT := 279; (* Manufacturer: Geometris LP | Location: Houston, TX USA - 2008-02-15 *)
    M_LEICA_GEOSYSTEMS_PTY : UINT := 280; (* Manufacturer: Leica Geosystems Pty Ltd | Location: Brisbane, Queensland Australia - 2008-02-18 *)
    M_PRECISION_GOVERNORS : UINT := 281; (* Manufacturer: Precision Governors LLC | Location: Rockford, IL USA - 2008-02-23 *)
    M_MEDALLION_INSTRUMENTATION_SYSTEMS : UINT := 282; (* Manufacturer: Medallion Instrumentation Systems | Location: Spring Lake, MI USA - 2008-03-14 *)
    M_CWF_HAMILTON_AND : UINT := 283; (* Manufacturer: CWF Hamilton & Co Ltd | Location: Christchurch, New Zealand - 2008-03-14 *)
    M_MOBILE_TECH_CHILE : UINT := 284; (* Manufacturer: Mobile Tech Chile | Location: Concepcion, Bio Bio Chile - 2008-05-11 *)
    M_SEA_RECOVERY : UINT := 285; (* Manufacturer: Sea Recovery Corp | Location: Rancho Dominguez, CA USA - 2008-05-11 *)
    M_COELMO_SRL : UINT := 286; (* Manufacturer: Coelmo srl | Location: Acerra, Italy - 2008-05-11 *)
    M_NTECH_INDUSTRIES_287 : UINT := 287; (* Manufacturer: NTech Industries, Inc | Location: Ukiah, CA USA - 2008-05-11 *)
    M_MITSUBISHI_FUSO_TRUCK_AND_BUS : UINT := 288; (* Manufacturer: Mitsubishi FUSO Truck & Bus Corp. | Location: Kawasaki, Kanagawa Japan - 2008-05-21 *)
    M_WATLOW : UINT := 289; (* Manufacturer: Watlow | Location: St. Louis, MO USA - 2008-05-21 *)
    M_KUEBLER : UINT := 290; (* Manufacturer: Kuebler GmbH | Location: VS-Schwenningen, Germany - 2008-07-12 *)
    M_GROENEVELD_TRANSPORT_EFFICIENCY_BV : UINT := 291; (* Manufacturer: Groeneveld Transport Efficiency BV | Location: Gorinchem, The Netherlands - *)
    M_IKUSI_ANGEL_IGLESIAS : UINT := 292; (* Manufacturer: IKUSI - Angel Iglesias S.A. | Location: San Sebastian, Guipuzcoa Spain - 2008-07-12 *)
    M_SPYDER_CONTROLS : UINT := 293; (* Manufacturer: Spyder Controls Corp. | Location: Lacombe, AB Canada - 2008-07-12 *)
    M_GRAYHILL : UINT := 294; (* Manufacturer: Grayhill Inc. | Location: LaGrange, IL USA - 2008-07-12 *)
    M_BEP_MARINE : UINT := 295; (* Manufacturer: BEP Marine | Location: Albany, North Shore City New Zealand - 2008-07-12 *)
    M_MICRO_DYNAMICS : UINT := 296; (* Manufacturer: micro dynamics GmbH | Location: Cologne, Germany - 2008-07-16 *)
    M_ZONAR_SYSTEMS : UINT := 297; (* Manufacturer: Zonar Systems Inc | Location: Seattle, WA USA - 2008-07-26 *)
    M_HOLLEY_PERFORMANCE : UINT := 298; (* Manufacturer: Holley Performance | Location: Bowling Green, KY USA - 2008-07-26 *)
    M_RAUCH : UINT := 299; (* Manufacturer: Rauch | Location: Sinzheim, Germany - 2008-08-11 *)
    M_SYSTRON_DONNER_AUTOMOTIVE : UINT := 300; (* Manufacturer: Systron Donner Automotive | Location: Concord, CA USA - 2008-08-11 *)
    M_PARKER_HANNIFIN_FDE_GROUP : UINT := 301; (* Manufacturer: Parker Hannifin (UK) Ltd FDE group | Location: Thetford, Norfolk UK - 2008-08-14 *)
    M_NISSIN_KOGYO : UINT := 302; (* Manufacturer: Nissin Kogyo Co., LTD | Location: Ueda-city, Nagano prefecture Japan - 2008-09-05 *)
    M_CTS : UINT := 303; (* Manufacturer: CTS Corporation | Location: Elkhart, IN USA - 2008-09-05 *)
    M_EMPIRBUS : UINT := 304; (* Manufacturer: EmpirBus AB | Location: Uddevalla, Sweden - 2008-09-05 *)
    M_NOVATEL : UINT := 305; (* Manufacturer: NovAtel Inc | Location: Calgary, AB Canada - 2008-09-20 *)
    M_SLEIPNER_MOTOR : UINT := 306; (* Manufacturer: Sleipner Motor AB | Location: Fredrikstad, Norway - 2008-09-20 *)
    M_MAS_TECHNOLOGIES : UINT := 307; (* Manufacturer: MAS Technologies | Location: Harleysville, PA USA - 2008-09-20 *)
    M_CYNTRX : UINT := 308; (* Manufacturer: Cyntrx | Location: De Pere, WI USA - 2008-10-31 *)
    M_KRAUSS_MAFFEI_WEGMANN_AND : UINT := 309; (* Manufacturer: Krauss-Maffei Wegmann GmbH & Co. KG | Location: Munich, Germany - 2008-10-31 *)
    M_TECNORD_SRL : UINT := 310; (* Manufacturer: TECNORD srl | Location: Modena, Italy - 2008-10-31 *)
    M_PATRICK_POWER_PRODUCTS : UINT := 311; (* Manufacturer: Patrick Power Products | Location: Elkridge, MD USA - 2008-11-09 *)
    M_LECTRONIX : UINT := 312; (* Manufacturer: Lectronix, Inc. | Location: Lansing, MI USA - 2008-11-20 *)
    M_ILMOR_ENGINEERING : UINT := 313; (* Manufacturer: Ilmor Engineering, Inc. | Location: Plymouth, MI USA - 2008-12-02 *)
    M_CSM : UINT := 314; (* Manufacturer: CSM GmbH | Location: Filderstadt, Germany - 2008-12-08 *)
    M_ICOM_INCORPORATED : UINT := 315; (* Manufacturer: Icom Incorporated | Location: Osaka, Japan - 2008-12-15 *)
    M_ITT_FLOW_CONTROL : UINT := 316; (* Manufacturer: ITT Flow Control | Location: Santa Ana, CA USA - 2008-12-18 *)
    M_NAVTRONICS_BVBA : UINT := 317; (* Manufacturer: Navtronics Bvba | Location: Geel, Belgium - 2009-01-19 *)
    M_SAT_PLAN : UINT := 318; (* Manufacturer: SAT Plan | Location: Beauvais Tillé, Oise France - 2009-01-19 *)
    M_CADEC_GLOBAL : UINT := 319; (* Manufacturer: Cadec Global | Location: Manchester, NH USA - 2009-01-19 *)
    M_MIEDEMA_LANDBOUWWERKTUIGENFABRIEK_B_V : UINT := 320; (* Manufacturer: Miedema Landbouwwerktuigenfabriek B.V. | Location: Winsum, The Netherlands - *)
    M_ULTRA_ELECTRONICS_ELECTRICS : UINT := 321; (* Manufacturer: Ultra Electronics, Electrics | Location: Cheltenham, UK - 2009-01-19 *)
    M_MICHENKA_S_R_O : UINT := 322; (* Manufacturer: MICHENKA s.r.o. | Location: Koprivnice, Czech Republic - 2009-01-19 *)
    M_MOBILEYE_VISION_TECHNOLOGIES : UINT := 323; (* Manufacturer: Mobileye Vision Technologies Ltd. | Location: Jerusalem, Israel - 2009-02-01 *)
    M_SNAP_ON_DIAGNOSTICS : UINT := 324; (* Manufacturer: Snap-on Diagnostics | Location: Lincolnshire, IL USA - 2009-02-01 *)
    M_ASM_AUTOMATION_SENSORIK_MESSTECHNIK : UINT := 325; (* Manufacturer: ASM Automation Sensorik Messtechnik GmbH | Location: Moosinning, Germany - *)
    M_AKRON_BRASS_COMPANY : UINT := 326; (* Manufacturer: Akron Brass Company | Location: Wooster, OH USA - 2009-02-12 *)
    M_SONCEBOZ : UINT := 327; (* Manufacturer: Sonceboz SA | Location: Sonceboz, Switzerland - 2009-02-12 *)
    M_QWERTY_ELECTRONIK : UINT := 328; (* Manufacturer: Qwerty Electronik AB | Location: Bagarmossen, Sweden - 2009-03-22 *)
    M_DEIF : UINT := 329; (* Manufacturer: Deif A/S | Location: Skive, Denmark - 2009-03-22 *)
    M_KIDDE_AEROSPACE_AND_DEFENSE : UINT := 330; (* Manufacturer: Kidde Aerospace and Defense | Location: Wilson, NC USA - 2009-03-22 *)
    M_HORTON : UINT := 331; (* Manufacturer: Horton, Inc. | Location: Roseville, MN USA - 2009-03-22 *)
    M_HWH : UINT := 332; (* Manufacturer: HWH Corporation | Location: Moscow, IA USA - 2009-04-10 *)
    M_LINK_MANUFACTURING : UINT := 333; (* Manufacturer: Link Manufacturing, Ltd. (formerly Hadley Products Corporation) | Location: Sioux *)
    M_TAKATA_PETRI_AG : UINT := 334; (* Manufacturer: Takata-Petri AG | Location: Aschaffenburg, Germany - 2009-04-19 *)
    M_EVO_ELECTRIC : UINT := 335; (* Manufacturer: Evo Electric Ltd | Location: Woking, Surrey, UK - 2009-05-15 *)
    M_APE_S_R_O : UINT := 336; (* Manufacturer: APE s.r.o. | Location: Bradlec, Czech Republic - 2009-05-18 *)
    M_CARRARO : UINT := 337; (* Manufacturer: Carraro S.p.A. | Location: Campodarsego, Italy - 2009-05-18 *)
    M_GRAF_SYTECO : UINT := 338; (* Manufacturer: GRAF-SYTECO | Location: Tuningen, Germany - 2009-06-21 *)
    M_COMPETENCE_CENTER_ISOBUS_E_V : UINT := 339; (* Manufacturer: Competence Center ISOBUS e.V. | Location: Osnabrück, Germany - 2015-07-27 *)
    M_CONTINENTAL_AG : UINT := 340; (* Manufacturer: Continental AG | Location: Hannover, Germany - 2009-06-24 *)
    M_BONING_AND : UINT := 341; (* Manufacturer: Boning GmbH & Co | Location: Ganderkesee, Germany - 2009-07-01 *)
    M_THOMAS_MAGNETE : UINT := 342; (* Manufacturer: THOMAS MAGNETE GmbH | Location: Herdorf, Germany - 2009-07-25 *)
    M_BAUMER_GROUP : UINT := 343; (* Manufacturer: Baumer Group | Location: Villingen-Schwenningen, Germany - 2009-07-25 *)
    M_PARVUS : UINT := 344; (* Manufacturer: Parvus Corporation | Location: Salt Lake City, UT USA - 2009-07-25 *)
    M_KOREAN_MARITIME_UNIVERSITY : UINT := 345; (* Manufacturer: Korean Maritime University | Location: Busan, Korea - 2009-07-25 *)
    M_CONTROL_SOLUTIONS : UINT := 346; (* Manufacturer: Control Solutions | Location: Aurora, IL USA - 2009-08-09 *)
    M_HONEYWELL : UINT := 347; (* Manufacturer: Honeywell | Location: Morristown, NJ USA - 2009-08-21 *)
    M_AMAZONEN_WERKE_H_DREYER : UINT := 348; (* Manufacturer: Amazonen Werke H. Dreyer | Location: Hasbergen, Germany - 2009-08-21 *)
    M_SUONENTIETO : UINT := 349; (* Manufacturer: Suonentieto | Location: Kuopio, Finland - 2009-08-21 *)
    M_NORIS_MARINE_SYSTEMS_AND : UINT := 350; (* Manufacturer: Noris Marine Systems GmbH & Co KG | Location: Nuremberg, Germany - 2009-08-21 *)
    M_THRANE_AND_THRANE : UINT := 351; (* Manufacturer: Thrane & Thrane | Location: Gentofte, Denmark - 2009-08-30 *)
    M_SAME_DEUTZ_FAHR_GROUP : UINT := 352; (* Manufacturer: SAME DEUTZ-FAHR GROUP S.p.A. | Location: Treviglio, Italy - 2015-07-27 *)
    M_HEGEMON_ELECTRONICS : UINT := 353; (* Manufacturer: Hegemon Electronics, Inc. | Location: Sterling Heights, MI USA - 2009-09-20 *)
    M_JUNKKARI_OY : UINT := 354; (* Manufacturer: Junkkari OY | Location: Yliharma, Finland - 2009-10-08 *)
    M_MASTERVOLT_INTERNATIONAL_B_V : UINT := 355; (* Manufacturer: Mastervolt International B.V. | Location: Amsterdam, The Netherlands - 2009-10-09 *)
    M_FISCHER_PANDA_GENERATORS : UINT := 356; (* Manufacturer: Fischer Panda Generators, Inc | Location: Oakland Park, FL USA - 2009-10-20 *)
    M_HARDI_INTERNATIONAL : UINT := 357; (* Manufacturer: Hardi International A/S | Location: Taastrup, Denmark - 2009-11-08 *)
    M_VICTRON_ENERGY_B_V : UINT := 358; (* Manufacturer: Victron Energy B.V. | Location: Almere-Haven, The Netherlands - 2009-11-08 *)
    M_LUDWIG_BERGMANN : UINT := 359; (* Manufacturer: Ludwig Bergmann GmbH | Location: Goldenstedt, Germany - 2009-11-08 *)
    M_HJS_EMISSION_TECHNOLOGY_AND : UINT := 360; (* Manufacturer: HJS Emission Technology GmbH & Co KG (formerly HJS Fahrzeugtechnik GmbH & Co KG) | *)
    M_INMACH : UINT := 361; (* Manufacturer: InMach | Location: Ulm, Germany - 2010-01-15 *)
    M_POETTINGER_LANDTECHNIK : UINT := 362; (* Manufacturer: Poettinger Landtechnik GmbH (formerly Alois Poettinger Maschinenfabrik GmbH) | *)
    M_BEI_DUNCAN : UINT := 363; (* Manufacturer: BEI Duncan | Location: Goleta, CA USA - 2010-01-30 *)
    M_OEM_CONTROLS : UINT := 364; (* Manufacturer: OEM Controls Inc. | Location: Shelton, CT USA - 2010-01-30 *)
    M_DIGI_STAR : UINT := 365; (* Manufacturer: Digi-Star, LLC | Location: Fort Atkinson, WI USA - 2010-01-30 *)
    M_VIEWNYX : UINT := 366; (* Manufacturer: Viewnyx Corp. | Location: Kanata, ON Canada - 2010-01-30 *)
    M_FLIEGL_AGRARTECHNIK : UINT := 367; (* Manufacturer: Fliegl Agrartechnik | Location: Muehldorf am Inn, Germany - 2013-09-12 *)
    M_HANSENHOF_ELECTRONIC : UINT := 368; (* Manufacturer: HANSENHOF_electronic | Location: Reifland, Germany - 2010-01-30 *)
    M_POWER_TORQUE_ENGINEERING : UINT := 369; (* Manufacturer: Power Torque Engineering Ltd | Location: Coventry, UK - 2010-02-14 *)
    M_ROLLS_ROYCE_MARINE : UINT := 370; (* Manufacturer: Rolls-Royce Marine AS | Location: Aalesund, Norway - 2010-05-15 *)
    M_HEINZMANN_AND : UINT := 371; (* Manufacturer: Heinzmann GmbH & Co. KG | Location: Schoenau, Germany - 2010-04-01 *)
    M_DELPHI : UINT := 372; (* Manufacturer: Delphi | Location: Auburn Hills, MI USA - 2010-04-01 *)
    M_ELECTRONIC_DESIGN : UINT := 373; (* Manufacturer: Electronic Design Inc. | Location: Sheboygan, WI USA - 2010-05-15 *)
    M_NORTHERN_LIGHTS : UINT := 374; (* Manufacturer: Northern Lights, Inc. | Location: Seattle, WA USA - 2010-05-15 *)
    M_WILLIAMS_CONTROLS : UINT := 375; (* Manufacturer: Williams Controls Inc. | Location: Portland, OR USA - 2010-05-15 *)
    M_QUAKE_GLOBAL : UINT := 376; (* Manufacturer: Quake Global | Location: San Diego, CA USA - 2010-06-15 *)
    M_IFM_ELECTRONIC : UINT := 377; (* Manufacturer: ifm electronic gmbh | Location: Essen, Germany - 2010-06-15 *)
    M_GLENDINNING_MARINE_PRODUCTS : UINT := 378; (* Manufacturer: Glendinning Marine Products | Location: Conway, SC USA - 2010-06-15 *)
    M_YAMABIKO : UINT := 379; (* Manufacturer: Yamabiko Corporation | Location: Iwate, Japan - 2010-06-20 *)
    M_SUNTECH_INTERNATIONAL : UINT := 380; (* Manufacturer: Suntech International Ltd. | Location: Seoul, Korea - 2010-06-20 *)
    M_B_AND_G : UINT := 381; (* Manufacturer: B & G | Location: Romsey, UK - 2010-08-20 *)
    M_NATIONAL_AGRICULTURE_AND_FOOD_RESEARCH_ORGANIZATION : UINT := 382; (* Manufacturer: National Agriculture and Food Research Organization | Location: Ibaraki, Japan - *)
    M_MCL_INDUSTRIES : UINT := 383; (* Manufacturer: MCL Industries | Location: Pulaski, WI USA - 2010-08-20 *)
    M_CAMANO_LIGHT : UINT := 384; (* Manufacturer: Camano Light | Location: Camano Island, WA USA - 2010-08-20 *)
    M_JOHNSON_OUTDOOR_MARINE_ELECTRONICS : UINT := 385; (* Manufacturer: Johnson Outdoor Marine Electronics | Location: Alpharetta, GA USA - 2010-08-20 *)
    M_JLG_AUTOMATION_BVBA : UINT := 386; (* Manufacturer: JLG Automation BVBA | Location: Gent, Belgium - 2010-08-20 *)
    M_ORSCHELN_PRODUCTS : UINT := 387; (* Manufacturer: Orscheln Products, LLC | Location: Moberly, MO USA - 2010-08-20 *)
    M_INNOMATIX : UINT := 388; (* Manufacturer: Innomatix, LLC | Location: Iowa City, IA USA - 2010-08-20 *)
    M_BENCHMARK_ELECTRONICS_MINNESOTA_DIVISION : UINT := 389; (* Manufacturer: Benchmark Electronics, Minnesota Division | Location: Rochester, MN USA - *)
    M_PARTECH : UINT := 390; (* Manufacturer: Partech Inc. | Location: Lake Orion, MI USA - 2010-08-20 *)
    M_ELECTRONIC_DESIGN_FOR_INDUSTRY : UINT := 391; (* Manufacturer: Electronic Design for Industry, Inc | Location: Belpre, OH USA - 2010-08-20 *)
    M_TIANYUAN_TECHNOLOGY : UINT := 392; (* Manufacturer: Tianyuan Technology Co Ltd. | Location: Shijiazhuang, China - 2010-08-28 *)
    M_HARVEST_TEC : UINT := 393; (* Manufacturer: Harvest Tec, Inc | Location: Hudson, WI USA - 2010-08-28 *)
    M_CAPI_2_NEDERLAND_B_V : UINT := 394; (* Manufacturer: Capi 2 Nederland B.V. | Location: Nuenen, The Netherlands - 2010-09-15 *)
    M_GENTEC_S_R_L : UINT := 395; (* Manufacturer: GENTEC S.R.L. | Location: Villa Constitucion, Argentina - 2010-09-20 *)
    M_BEYOND_MEASURE : UINT := 396; (* Manufacturer: Beyond Measure | Location: Appleton, WI USA - 2011-01-03 *)
    M_SANYO_KIKI : UINT := 397; (* Manufacturer: Sanyo-kiki Co Ltd. | Location: Okayama, Japan - 2010-10-30 *)
    M_HILITE_INTERNATIONAL : UINT := 398; (* Manufacturer: Hilite International | Location: Marktheidenfeld, Germany - 2010-10-30 *)
    M_ISEKI_AND : UINT := 399; (* Manufacturer: ISEKI & Co., Ltd. | Location: Ehime, Japan - 2010-11-01 *)
    M_LIVORSI_MARINE : UINT := 400; (* Manufacturer: Livorsi Marine | Location: Grayslake, IL USA - 2010-11-03 *)
    M_TORQEEDO : UINT := 401; (* Manufacturer: Torqeedo GmbH | Location: Stamberg, Germany - 2010-11-03 *)
    M_SIMMA_SOFTWARE : UINT := 402; (* Manufacturer: Simma Software, Inc. | Location: Terre Haute, IN USA - 2010-12-15 *)
    M_TRACKWELL_ADS : UINT := 403; (* Manufacturer: Trackwell ADS, Inc. | Location: Houston, TX USA - 2010-12-15 *)
    M_COM_NAV_MARINE : UINT := 404; (* Manufacturer: Com Nav Marine Ltd | Location: Richmond, BC Canada - 2010-12-15 *)
    M_WEMA_SYSTEM : UINT := 405; (* Manufacturer: Wema System AS | Location: Bergen, Norway - 2010-12-15 *)
    M_VECIMA_NETWORKS : UINT := 406; (* Manufacturer: Vecima Networks Inc. | Location: Saskatoon, SK Canada - 2010-12-15 *)
    M_COMTECH_MOBILE_DATACOM : UINT := 407; (* Manufacturer: Comtech Mobile Datacom | Location: Germantown, MD USA - 2010-12-15 *)
    M_CORVUS_ENERGY : UINT := 408; (* Manufacturer: Corvus Energy Ltd. | Location: Richmond, BC Canada - 2010-12-15 *)
    M_TRANSFLUID_S_R_L : UINT := 409; (* Manufacturer: Transfluid S.r.L. | Location: Gallarate, Italy - 2010-12-15 *)
    M_COBO_DIVISIONE_3B6 : UINT := 410; (* Manufacturer: COBO S.p.A. Divisione 3B6 | Location: Castelletto sopra Ticino, Italy - 2010-12-15 *)
    M_HY_DRIVE_TECHNOLOGIES : UINT := 411; (* Manufacturer: Hy-Drive Technologies Ltd. | Location: Mississauga, ON Canada - 2010-12-23 *)
    M_WEBTECH_WIRELESS : UINT := 412; (* Manufacturer: WebTech Wireless Inc. | Location: Burnaby, BC Canada - 2010-12-23 *)
    M_DATAPROSS_NIJBROEK_BV : UINT := 413; (* Manufacturer: Datapross Nijbroek bv | Location: Nijbroek, The Netherlands - 2011-01-04 *)
    M_CATTRON_GROUP_INTERNATIONAL : UINT := 414; (* Manufacturer: Cattron Group International | Location: Sharpsvillle, PA USA - 2011-01-06 *)
    M_VALID_MANUFACTURING : UINT := 415; (* Manufacturer: Valid Manufacturing Ltd. | Location: Salmon Arm, BC Canada - 2011-01-07 *)
    M_KUBOTA : UINT := 416; (* Manufacturer: Kubota Corporation | Location: Sakai, Japan - 2011-01-14 *)
    M_KZVALVE : UINT := 417; (* Manufacturer: KZValve | Location: Greenwood, NE USA - 2011-01-26 *)
    M_INTELLISTICK : UINT := 418; (* Manufacturer: Intellistick Inc | Location: Santa Ana, CA USA - 2011-01-26 *)
    M_FUSION_ELECTRONICS : UINT := 419; (* Manufacturer: Fusion Electronics Ltd | Location: Auckland, New Zealand - 2011-01-29 *)
    M_VERMEER_ACS_GROUP : UINT := 420; (* Manufacturer: Vermeer Corporation, ACS Group | Location: Pella, IA USA - 2011-01-31 *)
    M_VERTEX_STANDARD : UINT := 421; (* Manufacturer: Vertex Standard Co, Ltd | Location: Tokyo, Japan - 2011-02-11 *)
    M_TRUE_HEADING : UINT := 422; (* Manufacturer: True Heading AB | Location: Danderyd, Sweden - 2011-02-11 *)
    M_BSM_WIRELESS : UINT := 423; (* Manufacturer: BSM Wireless, Inc. | Location: Toronto, ON Canada - 2011-03-05 *)
    M_ODYNE : UINT := 424; (* Manufacturer: Odyne LLC | Location: Waukesha, WI USA - 2011-03-05 *)
    M_METHODE_ELECTRONICS_MDI : UINT := 425; (* Manufacturer: Methode Electronics Inc, MDI | Location: Chicago, IL USA - 2011-03-05 *)
    M_ROTA_ENGINEERING : UINT := 429; (* Manufacturer: Rota Engineering Ltd. | Location: Bury, Manchester, UK - 2011-04-27 *)
    M_AUTEQ_TELEMATICA : UINT := 430; (* Manufacturer: Auteq Telematica S.A. | Location: Sao Paulo, Brazil - 2011-04-27 *)
    M_TOHATSU : UINT := 431; (* Manufacturer: Tohatsu Corporation | Location: Tokyo, Japan - 2011-04-27 *)
    M_S_AND_A_SYSTEMS : UINT := 432; (* Manufacturer: S&A Systems, Inc. | Location: Rockwall, TX USA - 2011-04-27 *)
    M_ROWE_ELECTRONICS : UINT := 433; (* Manufacturer: Rowe Electronics | Location: Norwalk, IA USA - 2011-04-29 *)
    M_STORED_ENERGY_SYSTEMS : UINT := 434; (* Manufacturer: Stored Energy Systems | Location: Longmont, CO USA - 2011-04-29 *)
    M_ZUNHAMMER : UINT := 435; (* Manufacturer: Zunhammer GmbH | Location: Traunreut, Germany - 2011-05-06 *)
    M_KINZE_MANUFACTURING : UINT := 436; (* Manufacturer: Kinze Manufacturing | Location: Williamsburg, IA - 2011-05-18 *)
    M_DIGITAL_YACHT_LIMITED : UINT := 437; (* Manufacturer: Digital Yacht Limited | Location: Bristol, UK - 2011-05-18 *)
    M_COMAR_SYSTEMS : UINT := 438; (* Manufacturer: Comar Systems Ltd | Location: Cowes, Isle of Wight UK - 2011-05-18 *)
    M_HD_HYUNDAI : UINT := 439; (* Manufacturer: HD Hyundai (formerly Hyundai Heavy Industries) | Location: Ulsan, South Korea - *)
    M_CUMMINS_POWER_GENERATION : UINT := 440; (* Manufacturer: Cummins Power Generation | Location: Fridley, MN USA - 2011-06-18 *)
    M_PTG_REIFENDRUCKREGELSYSTEME : UINT := 441; (* Manufacturer: PTG Reifendruckregelsysteme GmbH | Location: Neuss, Germany - 2011-07-01 *)
    M_HORSCH_MASCHINEN_SE_AND : UINT := 442; (* Manufacturer: HORSCH Maschinen SE & Co. KG (formerly HORSCH Maschinen GmbH) | Location: *)
    M_SIGNALQUEST : UINT := 443; (* Manufacturer: SignalQuest, Inc. | Location: Lebanon, NH USA - 2011-07-01 *)
    M_ITT_POWER_SOLUTIONS : UINT := 444; (* Manufacturer: ITT Power Solutions | Location: West Springfield, MA USA - 2011-07-01 *)
    M_KAT_MECHATRONIC_ELECTRONIC_PRODUCT_DIVISION : UINT := 445; (* Manufacturer: KAT MECHATRONIC, Electronic Product Division | Location: Istanbul, Turkey - *)
    M_CERTTECH : UINT := 446; (* Manufacturer: CertTech, L.L.C. | Location: Lenexa, KS USA - 2011-07-29 *)
    M_GREAT_PLAINS_MFG : UINT := 447; (* Manufacturer: Great Plains Mfg. | Location: Salina, KS USA - 2011-07-29 *)
    M_STANADYNE_ELECTRONICS_SYSTEMS : UINT := 448; (* Manufacturer: Stanadyne Corporation, Electronics Systems | Location: Windsor, CT USA - 2011-08-09 *)
    M_POLARIS_INDUSTRIES : UINT := 449; (* Manufacturer: Polaris Industries Inc | Location: Medina, MN USA - 2011-08-22 *)
    M_DYCOR_TECHNOLOGIES : UINT := 450; (* Manufacturer: Dycor Technologies Ltd. | Location: Edmonton, AB Canada - 2011-08-22 *)
    M_PARKER_HANNIFIN : UINT := 451; (* Manufacturer: Parker Hannifin Corp | Location: Gardena, CA USA - 2011-08-22 *)
    M_WIKA_ALEXANDER_WIEGAND_SE_AND : UINT := 452; (* Manufacturer: WIKA Alexander Wiegand SE & Co. KG | Location: Klingenberg, Germany - 2011-10-15 *)
    M_COOPER_BUSSMANN : UINT := 453; (* Manufacturer: Cooper Bussmann | Location: Tualatin, OR USA - 2011-10-15 *)
    M_NGK_SPARK_PLUG : UINT := 454; (* Manufacturer: NGK Spark Plug Co. Ltd | Location: Komaki, Japan - 2011-10-15 *)
    M_ADZ_NAGANO : UINT := 455; (* Manufacturer: ADZ NAGANO GmbH | Location: Ottendorf-Okrilla, Germany - 2011-10-31 *)
    M_GENERAL_KINETICS : UINT := 456; (* Manufacturer: General Kinetics | Location: Manchester, NH USA - 2011-10-31 *)
    M_RUSELPROM_ELECTRICDRIVE : UINT := 457; (* Manufacturer: RUSELPROM-ElectricDrive Ltd | Location: Moscow, Russian Federation - 2011-10-31 *)
    M_CONTROL_SOLUTIONS_458 : UINT := 458; (* Manufacturer: Control Solutions, Inc. | Location: St. Paul, MN USA - 2011-10-31 *)
    M_ALLTEK_MARINE_ELECTRONICS : UINT := 459; (* Manufacturer: Alltek Marine Electronics Corp | Location: Neihu, Taiwan - 2011-11-06 *)
    M_SAN_GIORGIO_S_E_I_N : UINT := 460; (* Manufacturer: San Giorgio S.E.I.N. | Location: Genova, Italy - 2011-11-06 *)
    M_HAWE_HYDRAULIK_SE : UINT := 461; (* Manufacturer: HAWE Hydraulik SE | Location: Munich, Germany - 2011-11-13 *)
    M_IHI_SHIBAURA_MACHINERY : UINT := 462; (* Manufacturer: IHI Shibaura Machinery Corporation | Location: Matsumoto, Japan - 2011-11-13 *)
    M_PROBOTIQ : UINT := 463; (* Manufacturer: PROBOTIQ | Location: Cuijk, The Netherlands - 2012-01-02 *)
    M_LEACH_INTERNATIONAL : UINT := 464; (* Manufacturer: Leach International Corporation | Location: Buena Park, CA USA - 2012-01-02 *)
    M_ASHCROFT : UINT := 465; (* Manufacturer: Ashcroft Inc | Location: Stratford, CT USA - 2012-01-02 *)
    M_VEETHREE_ELECTRONICS_AND_MARINE : UINT := 466; (* Manufacturer: Veethree Electronics and Marine LLC | Location: Sarasota, FL USA - 2011-12-09 *)
    M_LELY_INDUSTRIES_N_V : UINT := 467; (* Manufacturer: Lely Industries N.V. | Location: Maassluis, The Netherlands - 2012-01-02 *)
    M_TYCO_FIRE_PROTECTION_PRODUCTS : UINT := 468; (* Manufacturer: Tyco Fire Protection Products | Location: Marinette, WI USA - 2012-01-02 *)
    M_RA_CONSULTING : UINT := 469; (* Manufacturer: RA Consulting GmbH | Location: Bruchsal, Germany - 2012-01-21 *)
    M_SI_TEX_MARINE_ELECTRONICS : UINT := 470; (* Manufacturer: SI-TEX Marine Electronics | Location: Riverhead, NY USA - 2012-01-21 *)
    M_SEA_CROSS_MARINE : UINT := 471; (* Manufacturer: Sea Cross Marine AB | Location: Udingo, Sweden - 2012-02-07 *)
    M_TENNECO : UINT := 472; (* Manufacturer: Tenneco Inc. | Location: Grass Lake, MI USA - 2012-02-07 *)
    M_BOSS_INDUSTRIES : UINT := 473; (* Manufacturer: Boss Industries, Inc. | Location: La Porte, IN USA - 2012-02-07 *)
    M_PERSEN_TECHNOLOGIES : UINT := 474; (* Manufacturer: Persen Technologies Inc. | Location: Winnipeg, MB Canada - 2012-02-07 *)
    M_GME : UINT := 475; (* Manufacturer: GME | Location: New South Wales, Australia - 2012-02-12 *)
    M_HUMMINGBIRD_MARINE_ELECTRONICS : UINT := 476; (* Manufacturer: Hummingbird Marine Electronics | Location: Alpharetta, GA USA - 2012-02-15 *)
    M_OILQUICK : UINT := 477; (* Manufacturer: OilQuick AB | Location: Hudiksvall, Sweden - 2012-02-17 *)
    M_OCEANSAT_B_V : UINT := 478; (* Manufacturer: OceanSat B.V. | Location: Nieuwendijk, The Netherlands - 2012-02-21 *)
    M_VAPOR_BUS_INTERNATIONAL : UINT := 479; (* Manufacturer: Vapor Bus International | Location: Buffalo Grove, IL USA - 2012-02-28 *)
    M_ENERDEL : UINT := 480; (* Manufacturer: EnerDel, Inc. | Location: Indianapolis, IN USA - 2012-02-29 *)
    M_CHETCO_DIGITAL_INSTRUMENTS : UINT := 481; (* Manufacturer: Chetco Digital Instruments | Location: Brookings, OR USA - 2012-03-12 *)
    M_TRICON_ELECTRONICS : UINT := 482; (* Manufacturer: Tricon Electronics | Location: Kolding, Denmark - 2012-03-12 *)
    M_VALEO : UINT := 483; (* Manufacturer: Valeo | Location: Creteil, France - 2012-04-13 *)
    M_HEADSIGHT : UINT := 484; (* Manufacturer: Headsight Inc. | Location: Bremen, IN USA - 2012-04-13 *)
    M_MATT_AUTOMOTIVE : UINT := 485; (* Manufacturer: MATT automotive | Location: Koscian, Poland - 2012-04-13 *)
    M_WESTPORT_INNOVATIONS : UINT := 486; (* Manufacturer: Westport Innovations Inc. | Location: Vancouver, BC Canada - 2012-04-13 *)
    M_DSE_TEST_SOLUTIONS : UINT := 487; (* Manufacturer: DSE Test Solutions A/S | Location: Horsens, Denmark - 2012-04-13 *)
    M_THE_CHARLES_MACHINE_WORKS : UINT := 488; (* Manufacturer: The Charles Machine Works, Inc. | Location: Perry, OK USA - 2012-04-16 *)
    M_APPAREO_SYSTEMS : UINT := 489; (* Manufacturer: Appareo Systems, LLC | Location: Fargo, ND USA - 2013-09-12 *)
    M_QUIKQ : UINT := 490; (* Manufacturer: QuikQ | Location: Franklin, TN USA - 2012-04-23 *)
    M_PENNY_AND_GILES : UINT := 491; (* Manufacturer: Penny and Giles Ltd | Location: Wales, UK - 2012-04-27 *)
    M_INERGY_AUTOMOTIVE_SYSTEMS : UINT := 492; (* Manufacturer: Inergy Automotive Systems | Location: Troy, MI USA - 2012-05-03 *)
    M_WATCHEYE : UINT := 493; (* Manufacturer: Watcheye | Location: Gouda, The Netherlands - 2012-05-03 *)
    M_SYNERJECT : UINT := 494; (* Manufacturer: Synerject | Location: Toulouse, France - 2012-05-03 *)
    M_HOLMER_MASCHINENBAU : UINT := 495; (* Manufacturer: HOLMER Maschinenbau GmbH | Location: Schierling, Germany - 2012-05-03 *)
    M_W_GESSMANN : UINT := 496; (* Manufacturer: W. Gessmann GmbH | Location: Leingarten, Germany - 2012-06-01 *)
    M_SENTRON_SISTEMAS_EMBARCADOS : UINT := 497; (* Manufacturer: SENTRON Sistemas Embarcados | Location: Sao Carlos, Brazil - 2012-06-01 *)
    M_INNOVATIVE_DESIGN_SOLUTIONS : UINT := 498; (* Manufacturer: Innovative Design Solutions, Inc. | Location: Troy, MI USA - 2012-06-01 *)
    M_LCJ_CAPTEURS : UINT := 499; (* Manufacturer: LCJ Capteurs | Location: Vertou, France - 2012-07-10 *)
    M_OXBO_INTERNATIONAL : UINT := 500; (* Manufacturer: Oxbo International Corporation | Location: Byron, NY USA - 2012-07-12 *)
    M_AGROTRONIX : UINT := 501; (* Manufacturer: Agrotronix S.A. | Location: Douvrin, France - 2012-07-18 *)
    M_ATTWOOD : UINT := 502; (* Manufacturer: Attwood Corporation | Location: Lowell, MI USA - 2012-08-17 *)
    M_NAVIOP_S_R_L : UINT := 503; (* Manufacturer: Naviop S.R.L. | Location: Forli, Italy - 2012-08-30 *)
    M_VESPER_MARINE : UINT := 504; (* Manufacturer: Vesper Marine | Location: Auckland, New Zealand - 2012-09-25 *)
    M_YETTER_FARM_EQUIPMENT : UINT := 505; (* Manufacturer: Yetter Farm Equipment | Location: Colchester, IL USA - 2012-09-25 *)
    M_IHI_STAR_MACHINERY : UINT := 506; (* Manufacturer: IHI STAR Machinery Corporation | Location: Hokkaido, Japan - 2012-09-25 *)
    M_ISOBUS_TEST_CENTER : UINT := 507; (* Manufacturer: ISOBUS Test Center | Location: Osnabrück, Germany - 2015-07-27 *)
    M_TRANSTECH_INNOVATIONS : UINT := 508; (* Manufacturer: Transtech Innovations | Location: Varennes, QC Canada - 2012-10-26 *)
    M_MOTORTECH : UINT := 509; (* Manufacturer: MOTORTECH GmbH | Location: Celle, Germany - 2012-10-26 *)
    M_MARINESOFT : UINT := 510; (* Manufacturer: Marinesoft Co. Ltd | Location: Busan, South Korea - 2012-10-26 *)
    M_SULKY : UINT := 511; (* Manufacturer: Sulky | Location: Chateaubourg, France - 2012-10-26 *)
    M_INPOWER : UINT := 512; (* Manufacturer: Inpower LLC | Location: Lewis Center, OH USA - 2012-11-01 *)
    M_PRECISION_TECHNOLOGY : UINT := 513; (* Manufacturer: Precision Technology | Location: Toowoomba, QLD Australia - 2019-11-12 *)
    M_DISTEK_INTEGRATION : UINT := 514; (* Manufacturer: DISTek Integration, Inc. | Location: Cedar Falls, IA USA - 2012-11-10 *)
    M_GINAF_TRUCKS_NEDERLAND_B_V : UINT := 515; (* Manufacturer: GINAF Trucks Nederland B.V. | Location: Veenendaal, The Netherlands - 2012-11-14 *)
    M_AVAT_AUTOMATION : UINT := 516; (* Manufacturer: AVAT Automation GmbH | Location: Tuebingen, Germany - 2012-11-30 *)
    M_NOLAND_ENGINEERING : UINT := 517; (* Manufacturer: Noland Engineering | Location: Melbourne, FL USA - 2012-12-06 *)
    M_TRANSAS_USA : UINT := 518; (* Manufacturer: Transas USA Inc. | Location: Bothell, WA USA - 2012-12-06 *)
    M_PEETERS_LANDBOUWMACHINES_B_V : UINT := 519; (* Manufacturer: Peeters Landbouwmachines b.v. | Location: Etten-Leur, The Netherlands - 2012-12-12 *)
    M_TRAPEZE : UINT := 520; (* Manufacturer: Trapeze | Location: Cedar Rapids, IA USA - 2012-12-14 *)
    M_CLEVER_DEVICES : UINT := 521; (* Manufacturer: Clever Devices Ltd. | Location: Woodbury, NY USA - 2013-02-15 *)
    M_NEBRASKA_TRACTOR_TEST_LABORATORY : UINT := 522; (* Manufacturer: Nebraska Tractor Test Laboratory | Location: Lincoln, NE USA - 2013-02-15 *)
    M_REGGIO_EMILIA_INNOVAZIONE : UINT := 523; (* Manufacturer: Reggio Emilia Innovazione | Location: Reggio Emilia Italy - 2013-02-15 *)
    M_VOMAX_INSTRUMENTATION_PTY : UINT := 524; (* Manufacturer: Vomax Instrumentation Pty. Ltd. | Location: Marleston, SA Australia - 2013-02-21 *)
    M_RUST_SALES : UINT := 525; (* Manufacturer: Rust Sales INC | Location: Harwood, ND USA - 2013-02-26 *)
    M_LOFA_INDUSTRIES : UINT := 526; (* Manufacturer: LOFA Industries, Inc | Location: Roswell, GA USA - 2013-02-26 *)
    M_GKN_WALTERSCHEID : UINT := 527; (* Manufacturer: GKN Walterscheid GmbH | Location: Lohmar, Germany - 2013-02-27 *)
    M_HOGANAS_ELECTRIC_DRIVE_SYSTEMS : UINT := 528; (* Manufacturer: Hoganas AB, Electric Drive Systems | Location: Hoganas, Sweden - 2013-03-12 *)
    M_NATIONAL_INSTRUMENTS_KOREA : UINT := 529; (* Manufacturer: National Instruments Korea | Location: Seoul, South Korea - 2013-03-12 *)
    M_NMEA : UINT := 530; (* Manufacturer: NMEA | Location: Severna Park, MD USA - 2013-03-12 *)
    M_GENGE_AND_THOMA_AG : UINT := 531; (* Manufacturer: Genge & Thoma AG | Location: Bern, Switzerland - 2013-03-28 *)
    M_ONWA_MARINE_ELECTRONICS : UINT := 532; (* Manufacturer: Onwa Marine Electronics Co Ltd. | Location: Hong Kong, China - 2013-03-28 *)
    M_DORAN_MANUFACTURING : UINT := 533; (* Manufacturer: Doran Manufacturing, LLC | Location: Cincinnati, OH USA - 2013-04-14 *)
    M_WEBASTO_THERMO_AND_COMFORT_SE : UINT := 534; (* Manufacturer: Webasto Thermo & Comfort SE | Location: Gilching, Germany - 2013-04-14 *)
    M_MOTORPAL_A_S : UINT := 535; (* Manufacturer: MOTORPAL, a.s. | Location: Jihlava, Czech Republic - 2013-04-14 *)
    M_SSI_TECHNOLOGIES : UINT := 536; (* Manufacturer: SSI Technologies | Location: Janesville, WI USA - 2013-04-25 *)
    M_SCHRADER_ELECTRONICS : UINT := 537; (* Manufacturer: Schrader Electronics Ltd. | Location: Antrim, N. Ireland - 2013-04-25 *)
    M_CROP_VENTURES : UINT := 538; (* Manufacturer: Crop Ventures, Inc. | Location: Omaha, NE USA - 2013-04-25 *)
    M_MOBILEVIEW : UINT := 539; (* Manufacturer: Mobileview | Location: Costa Mesa, CA USA - 2013-04-25 *)
    M_DINEX : UINT := 540; (* Manufacturer: Dinex A/S | Location: Middelfart, Denmark - 2013-04-25 *)
    M_TOTAL_FIRE_SYSTEMS : UINT := 541; (* Manufacturer: Total Fire Systems, Inc. | Location: Youngsville, NC USA - 2013-04-25 *)
    M_DINAMICA_GENERALE : UINT := 542; (* Manufacturer: Dinamica Generale s.p.a. | Location: Poggio Rusco, Italy - 2013-05-08 *)
    M_BAUER_MASCHINEN : UINT := 543; (* Manufacturer: BAUER Maschinen GmbH | Location: Schrobenhausen, Germany - 2013-05-23 *)
    M_AU_GROUP_ELECTRONICS : UINT := 544; (* Manufacturer: Au Group Electronics | Location: Windsor, ON Canada - 2013-05-23 *)
    M_GS_GLOBAL_RESOURCES : UINT := 545; (* Manufacturer: GS Global Resources (formerly GS Hydraulics) | Location: Mukwonago, WI USA - *)
    M_MARUYAMA_MFG : UINT := 546; (* Manufacturer: Maruyama Mfg Co, Inc. | Location: Togane, Chiba, Japan - 2013-06-11 *)
    M_THOMSON_LINEAR : UINT := 547; (* Manufacturer: Thomson Linear LLC | Location: Marengo, IL USA - 2013-06-17 *)
    M_TM4 : UINT := 548; (* Manufacturer: TM4 Inc. | Location: Boucherville, QC Canada - 2013-06-28 *)
    M_ROAD_DEUTSCHLAND : UINT := 549; (* Manufacturer: ROAD Deutschland GmbH | Location: Bretten, Germany - 2013-06-28 *)
    M_SUN_A : UINT := 550; (* Manufacturer: SUN-A Corporation | Location: Hiroshima, Japan - 2013-07-17 *)
    M_WEXLER_CSD : UINT := 551; (* Manufacturer: Wexler CSD Ltd. | Location: Rishon LeZion, Israel - 2013-07-17 *)
    M_MATSUYAMA_PLOW_MFG : UINT := 552; (* Manufacturer: Matsuyama Plow Mfg Co, Ltd | Location: Nagano, Japan - 2013-07-23 *)
    M_KIB_ELECTRONICS : UINT := 553; (* Manufacturer: KIB Electronics | Location: Elkhart, IN USA - 2013-08-11 *)
    M_IRIS_INFRARED_AND_INTELLIGENT_SENSORS : UINT := 554; (* Manufacturer: iris-GmbH infrared & intelligent sensors | Location: Berlin, Germany - 2013-08-20 *)
    M_SASAKI : UINT := 555; (* Manufacturer: Sasaki Corporation | Location: Towada City, Japan - 2013-08-21 *)
    M_HD_HYUNDAI_INFRACORE_NORWAY : UINT := 556; (* Manufacturer: HD Hyundai Infracore Norway (formerly Doosan Infracore Norway) | Location: *)
    M_ROCKSON_AUTOMATION : UINT := 557; (* Manufacturer: Rockson Automation GmbH | Location: Kiel, Germany - 2013-09-12 *)
    M_DAVIS_INSTRUMENTS : UINT := 558; (* Manufacturer: Davis Instruments Corp. | Location: Hayward, CA USA - 2013-10-12 *)
    M_FOUR_PEAKS_NAVIGATION : UINT := 559; (* Manufacturer: Four Peaks Navigation | Location: Overgaard, AZ USA - 2013-10-12 *)
    M_IOWA_STATE_UNIVERSITY_AGRICULTURAL_AND_BIOSYSTEMS_ENGINEERING : UINT := 560; (* Manufacturer: Iowa State University, Agricultural and Biosystems Engineering | Location: Ames, IA *)
    M_B_PLUS : UINT := 561; (* Manufacturer: b-plus GmbH | Location: Deggendorf, Germany - 2013-10-25 *)
    M_BOMBARDIER_TRANSPORTATION : UINT := 562; (* Manufacturer: Bombardier Transportation GmbH | Location: Mannheim, Germany - 2013-10-25 *)
    M_LOHR_SISTEMAS_ELETRONICOS_LTDA : UINT := 563; (* Manufacturer: LOHR Sistemas Eletronicos LTDA | Location: Caxias do Sul, Brazil - 2013-10-31 *)
    M_AUTO_POWER_ELECTRONIC : UINT := 564; (* Manufacturer: Auto Power Electronic | Location: Opole, Poland - 2013-11-01 *)
    M_MICRO_TRAK_SYSTEMS : UINT := 565; (* Manufacturer: Micro-Trak Systems, Inc. | Location: Eagle Lake, MN USA - 2013-11-12 *)
    M_GEODE_TECHNOLOGY : UINT := 566; (* Manufacturer: Geode Technology, Inc. | Location: Fredericton, NB Canada - 2013-11-13 *)
    M_LITHIUMSTART : UINT := 567; (* Manufacturer: Lithiumstart LLC | Location: Healdsburg, CA USA - 2013-11-26 *)
    M_MAKERSAN : UINT := 568; (* Manufacturer: Makersan Ltd. Co. | Location: Gebze, Turkey - 2013-11-26 *)
    M_LORD_MICROSTRAIN_SENSING_SYSTEMS : UINT := 569; (* Manufacturer: LORD MicroStrain Sensing Systems | Location: Willison, VT USA - 2013-12-16 *)
    M_FRENZEL_BERG_ELECTRONIC_AND : UINT := 570; (* Manufacturer: frenzel + berg electronic GmbH & Co. KG | Location: Ulm, Germany - 2014-01-04 *)
    M_MARINECRAFT : UINT := 571; (* Manufacturer: Marinecraft Co., Ltd. | Location: Pusan, South Korea - 2014-01-04 *)
    M_FASSE_VALVES : UINT := 572; (* Manufacturer: Fasse Valves | Location: Kearney, NE USA - 2014-01-04 *)
    M_OROLIA : UINT := 573; (* Manufacturer: Orolia Ltd | Location: Portsmouth, Hampshire UK - 2014-01-07 *)
    M_VISHAY_PRECISION_GROUP : UINT := 574; (* Manufacturer: Vishay Precision Group | Location: Bradford, West Yorkshire UK - 2014-01-13 *)
    M_LYTX : UINT := 575; (* Manufacturer: Lytx | Location: San Diego, CA USA - 2014-01-14 *)
    M_VECTIA : UINT := 576; (* Manufacturer: Vectia | Location: Irura, Guipuzcoa Spain - 2014-01-19 *)
    M_DENCHI_POWER : UINT := 577; (* Manufacturer: Denchi Power Ltd (formerly ABSL Power Solutions Limited) | Location: Thurso, *)
    M_ADVANSEA : UINT := 578; (* Manufacturer: advanSea | Location: Loriant, France - 2014-01-30 *)
    M_KVH_INDUSTRIES : UINT := 579; (* Manufacturer: KVH Industries, Inc. | Location: Middletown, RI USA - 2014-01-30 *)
    M_SAN_JOSE_TECHNOLOGY : UINT := 580; (* Manufacturer: San Jose Technology, Inc. | Location: New Taipei City, Taiwan - 2014-01-30 *)
    M_V_DERSTAD : UINT := 581; (* Manufacturer: Väderstad AB | Location: Väderstad, Sweden - 2022-06-15 *)
    M_INNOVATIVE_SOFTWARE_ENGINEERING : UINT := 582; (* Manufacturer: Innovative Software Engineering | Location: Coralville, IA USA - 2014-02-14 *)
    M_YACHTCONTROL : UINT := 583; (* Manufacturer: Yachtcontrol | Location: Hattern, The Netherlands - 2014-03-17 *)
    M_CARMEDIALAB : UINT := 584; (* Manufacturer: CarMedialab GmbH | Location: Bruchsal, Germany - 2014-03-24 *)
    M_INDUSTRIAL_ELECTRONIC_CONTROLS : UINT := 585; (* Manufacturer: Industrial Electronic Controls | Location: Rockford, IL USA - 2014-03-25 *)
    M_SUZUKI_MOTOR : UINT := 586; (* Manufacturer: Suzuki Motor Corp | Location: Hamamatsu, Japan - 2014-03-25 *)
    M_JCA_ELECTRONICS : UINT := 587; (* Manufacturer: JCA Electronics | Location: Winnipeg, MB Canada - 2014-03-27 *)
    M_VIGNAL_SYSTEMS : UINT := 588; (* Manufacturer: Vignal Systems | Location: Venissieux, France - 2014-03-28 *)
    M_MICO : UINT := 589; (* Manufacturer: MICO, Inc. | Location: North Mankato, MN USA - 2014-04-01 *)
    M_ARGO_HYTOS : UINT := 590; (* Manufacturer: ARGO-HYTOS GMBH | Location: Kraichtal, Germany - 2014-04-09 *)
    M_UNITED_STATES_COAST_GUARD : UINT := 591; (* Manufacturer: United States Coast Guard | Location: New London, CT USA - 2014-04-09 *)
    M_TECSIS : UINT := 592; (* Manufacturer: tecsis GmbH | Location: Offenbach, Germany - 2014-04-16 *)
    M_SENSATA_TECHNOLOGIES : UINT := 593; (* Manufacturer: Sensata Technologies | Location: Attleboro, MA USA - 2014-04-17 *)
    M_KONGSBERG_AUTOMOTIVE : UINT := 594; (* Manufacturer: Kongsberg Automotive | Location: Kongsberg, Norway - 2014-04-17 *)
    M_CUSTOMWARE : UINT := 595; (* Manufacturer: CustomWare | Location: Assen, The Netherlands - 2014-04-28 *)
    M_BRUNELCO_ELECTRONIC_INNOVATORS_B_V : UINT := 596; (* Manufacturer: Brunelco Electronic Innovators B.V. | Location: Haaksbergen, The Netherlands - *)
    M_HYDAC_FILTER_SYSTEMS : UINT := 597; (* Manufacturer: Hydac Filter Systems GmbH | Location: Sulzbach/Saar, Germany - 2014-05-23 *)
    M_ABB_TURBO_SYSTEMS : UINT := 598; (* Manufacturer: ABB Turbo Systems Ltd | Location: Baden, Switzerland - 2014-05-23 *)
    M_SPUDNIK_EQUIPMENT : UINT := 599; (* Manufacturer: Spudnik Equipment Co, LLC | Location: Blackfoot, ID USA - 2014-05-23 *)
    M_AQUATIC_AV : UINT := 600; (* Manufacturer: Aquatic AV | Location: San Jose, CA USA - 2014-05-23 *)
    M_NAVITAS_SYSTEMS : UINT := 601; (* Manufacturer: Navitas Systems | Location: Woodridge, IL USA - 2014-05-23 *)
    M_NOMAD_DIGITAL : UINT := 602; (* Manufacturer: Nomad Digital Ltd. | Location: Newcastle upon Tyne, UK - 2014-06-10 *)
    M_KEREVAL : UINT := 603; (* Manufacturer: Kereval | Location: Thorigne Fouillard, France - 2014-06-18 *)
    M_ROTOTILT_GROUP : UINT := 604; (* Manufacturer: Rototilt Group AB (formerly Indexator Rototilt Systems AB) | Location: Vindeln, *)
    M_AVENTICS : UINT := 605; (* Manufacturer: Aventics GmbH | Location: Laatzen, Germany - 2014-07-11 *)
    M_INTELLIAN_TECHNOLOGIES : UINT := 606; (* Manufacturer: Intellian Technologies | Location: Irvine, CA USA - 2014-07-11 *)
    M_KNAPPCO_CIVACON : UINT := 607; (* Manufacturer: Knappco/Civacon | Location: Kansas City, MO USA - 2014-07-15 *)
    M_GALE_BANKS_ENGINEERING : UINT := 608; (* Manufacturer: Gale Banks Engineering | Location: Azusa, CA USA - 2014-07-30 *)
    M_WALVOIL : UINT := 609; (* Manufacturer: Walvoil S.p.A. | Location: Reggio Emilia, Italy - 2014-07-30 *)
    M_TRAIL_TECH : UINT := 610; (* Manufacturer: Trail Tech | Location: Battle Ground, WA USA - 2014-07-30 *)
    M_ESTERLINE : UINT := 611; (* Manufacturer: Esterline | Location: Coeur d'Alene, ID USA - 2014-07-30 *)
    M_SAMWON_IT : UINT := 612; (* Manufacturer: Samwon IT | Location: Busan, Korea - 2014-08-04 *)
    M_HKS : UINT := 613; (* Manufacturer: HKS Co., Ltd. | Location: Shizuoka, Japan - 2014-08-21 *)
    M_ARLT_TECHNOLOGIES : UINT := 614; (* Manufacturer: ARLT Technologies GmbH | Location: Netphen, Germany - 2014-08-28 *)
    M_NETWORKFLEET_VERIZON_TELEMATICS : UINT := 615; (* Manufacturer: Networkfleet, Verizon Telematics | Location: San Diego, CA USA - 2014-08-28 *)
    M_SMART_TEC_S_R_O : UINT := 616; (* Manufacturer: SMART-TEC s.r.o. | Location: Velke Porici, Czech Republic - 2014-09-07 *)
    M_ZERO_EMISSION_VEHICLES : UINT := 617; (* Manufacturer: Zero Emission Vehicles | Location: Palmerston North, New Zealand - 2014-09-07 *)
    M_EVRARD : UINT := 618; (* Manufacturer: Evrard SA | Location: Beaurainville, France - 2014-09-16 *)
    M_RIGHT_WEIGH_LOAD_SCALES : UINT := 619; (* Manufacturer: Right Weigh Load Scales | Location: Sherwood, OR USA - 2014-09-16 *)
    M_BORGWARNER : UINT := 620; (* Manufacturer: BorgWarner Inc. (formerly Sevcon Ltd.) | Location: Auburn Hills, MI USA - *)
    M_HAGIE_MANUFACTURING_COMPANY : UINT := 621; (* Manufacturer: Hagie Manufacturing Company | Location: Clarion, IA USA - 2014-09-29 *)
    M_FLOYD_BELL : UINT := 622; (* Manufacturer: Floyd Bell Inc | Location: Columbus, OH USA - 2014-10-06 *)
    M_XIRGO_TECHNOLOGIES : UINT := 623; (* Manufacturer: Xirgo Technologies | Location: Camarillo, CA USA - 2014-10-08 *)
    M_BLACKBOX_MACHINE_CONTROL_PTY : UINT := 624; (* Manufacturer: Blackbox Machine Control Pty Ltd | Location: Maida Vale, WA Australia - 2014-10-11 *)
    M_GLOBAL_MRV : UINT := 625; (* Manufacturer: Global MRV Inc. | Location: Buffalo, NY USA - 2014-10-14 *)
    M_AVL_DITEST : UINT := 626; (* Manufacturer: AVL DiTEST GmbH | Location: Fuerth, Germany - 2014-10-21 *)
    M_RADIO_OCEAN : UINT := 627; (* Manufacturer: Radio Ocean | Location: Merignac, France - 2014-10-27 *)
    M_FALCK_SCHMIDT_DEFENCE_SYSTEMS : UINT := 628; (* Manufacturer: Falck Schmidt Defence Systems | Location: Odense C, Denmark - 2014-10-27 *)
    M_AGRI_INFO_DESIGN : UINT := 629; (* Manufacturer: Agri Info Design, Ltd. | Location: Hokkaido, Japan - 2014-10-29 *)
    M_SMARTDRIVE_SYSTEMS : UINT := 630; (* Manufacturer: SmartDrive Systems Inc. | Location: San Diego, CA USA - 2014-10-29 *)
    M_RELTIMA : UINT := 631; (* Manufacturer: Reltima | Location: Woburn, MA USA - 2014-11-09 *)
    M_PEPPERL_FUCHS : UINT := 632; (* Manufacturer: Pepperl+Fuchs GmbH | Location: Mannheim, Germany - 2014-11-25 *)
    M_TORC_ROBOTICS : UINT := 633; (* Manufacturer: TORC Robotics | Location: Blacksburg, VA USA - 2014-11-25 *)
    M_ROCKY_RESEARCH : UINT := 634; (* Manufacturer: Rocky Research | Location: Huntsville, AL USA - 2014-12-09 *)
    M_ARGO_TRACTORS : UINT := 635; (* Manufacturer: Argo Tractors S.p.A. | Location: Reggio Emilia, Italy - 2014-12-09 *)
    M_DIVELBISS : UINT := 636; (* Manufacturer: Divelbiss Corporation | Location: Fredericktown, OH USA - 2014-12-09 *)
    M_BAVARIA_YACHTBAU : UINT := 637; (* Manufacturer: Bavaria Yachtbau GmbH | Location: Giebelstadt, Germany - 2014-12-09 *)
    M_KVH_INDUSTRIES_638 : UINT := 638; (* Manufacturer: KVH Industries, Inc. | Location: Middletown, RI USA - 2015-01-06 *)
    M_STARTEC_S_R_L : UINT := 639; (* Manufacturer: Startec s.r.l. | Location: Sesto al Reghena (PN), Italy - 2015-01-06 *)
    M_POWER_SOLUTIONS_INTERNATIONAL : UINT := 640; (* Manufacturer: Power Solutions International | Location: Wood Dale, IL USA - 2015-01-12 *)
    M_DIVERSE_YACHT_SERVICES : UINT := 641; (* Manufacturer: Diverse Yacht Services | Location: Southampton, Hampshire UK - 2015-01-16 *)
    M_MOOG_ASPEN_MOTION_TECHNOLOGIES : UINT := 642; (* Manufacturer: Moog / Aspen Motion Technologies | Location: Radford, VA USA - 2015-01-22 *)
    M_BOGBALLE : UINT := 643; (* Manufacturer: Bogballe A/S | Location: Uldum, Denmark - 2015-01-22 *)
    M_KUS_USA : UINT := 644; (* Manufacturer: KUS USA | Location: Ft. Lauderdale, FL USA - 2015-01-22 *)
    M_ESD_ELECTRONIC_SYSTEM_DESIGN : UINT := 645; (* Manufacturer: esd electronic system design gmbh | Location: Hannover, Germany - 2015-01-22 *)
    M_VEENHUIS_MACHINES_B_V : UINT := 646; (* Manufacturer: Veenhuis Machines B.V. | Location: Raalte, The Netherlands - 2015-01-22 *)
    M_SILOKING : UINT := 647; (* Manufacturer: Siloking | Location: Tittmoning, Germany - 2015-01-22 *)
    M_OJSC_EKRAN : UINT := 648; (* Manufacturer: OJSC Ekran | Location: Borisov, Belarus - 2015-02-01 *)
    M_CONTROL_Q_B_V : UINT := 649; (* Manufacturer: Control-Q B.V. | Location: Vaassen, The Netherlands - 2015-02-10 *)
    M_SEIKO_EPSON : UINT := 650; (* Manufacturer: Seiko Epson Corp. | Location: Nagano, Japan - 2015-02-10 *)
    M_TAKAKITA : UINT := 651; (* Manufacturer: Takakita Co, Ltd. | Location: Nabari, Japan - 2015-02-10 *)
    M_MICROCONTROL_AND : UINT := 652; (* Manufacturer: MicroControl GmbH & Co. KG | Location: Troisdorf, Germany - 2015-02-12 *)
    M_AEV_SPOL_S_R_O : UINT := 653; (* Manufacturer: AEV, spol. s r. o. | Location: Kromeriz, Czech Republic - 2015-02-12 *)
    M_KOHLER_POWER_SYSTEMS_DETROIT_ENGINE_DEVELOPMENT_CENTER : UINT := 654; (* Manufacturer: Kohler Power Systems, Detroit Engine Development Center (DEDC) | Location: Detroit, *)
    M_GENGE_AND_THOMA_AG_655 : UINT := 655; (* Manufacturer: Genge & Thoma AG | Location: Lengnau, Switzerland - 2015-03-03 *)
    M_PRO_SOLUS_DO_BRASIL : UINT := 656; (* Manufacturer: PRO SOLUS do Brasil | Location: Campo Mourão, Brazil - 2015-03-03 *)
    M_TERZO_POWER_SYSTEMS : UINT := 657; (* Manufacturer: Terzo Power Systems | Location: Sacramento, CA USA - 2015-03-05 *)
    M_SHENZHEN_JIUZHOU_HIMUNICATION_TECHNOLOGY : UINT := 658; (* Manufacturer: Shenzhen Jiuzhou Himunication Technology Co., Ltd | Location: Shenzhen, China - *)
    M_DATA_PANEL : UINT := 659; (* Manufacturer: Data Panel Corp. | Location: Plymouth, MN USA - 2015-03-17 *)
    M_AUTO_GAZ_CENTRUM : UINT := 660; (* Manufacturer: Auto-Gaz Centrum | Location: Radom, Poland - 2015-03-30 *)
    M_SPAL_AUTOMOTIVE_S_R_L : UINT := 661; (* Manufacturer: SPAL Automotive S.r.l. | Location: Correggio, Italy - 2015-03-31 *)
    M_KISSLING_ELEKTROTECHNIK : UINT := 662; (* Manufacturer: Kissling Elektrotechnik GmbH | Location: Wildberg, Germany - 2015-03-31 *)
    M_DELTA_SYSTEMS : UINT := 663; (* Manufacturer: Delta Systems, Inc | Location: Streetsboro, OH USA - 2015-04-01 *)
    M_LEVEL_DEVELOPMENTS : UINT := 664; (* Manufacturer: Level Developments Ltd | Location: Croydon, Surrey UK - 2015-04-09 *)
    M_GEBR_BODE_AND : UINT := 665; (* Manufacturer: Gebr. Bode GmbH & Co. KG | Location: Kassel, Germany - 2015-04-13 *)
    M_SCHAEFFLER_TECHNOLOGIES_AG_AND : UINT := 666; (* Manufacturer: Schaeffler Technologies AG & Co., KG | Location: Herzogenaurach, Germany - *)
    M_BARTEC : UINT := 667; (* Manufacturer: Bartec | Location: Gotteszell, Germany - 2015-04-24 *)
    M_MACDON_INDUSTRIES : UINT := 668; (* Manufacturer: MacDon Industries Ltd. | Location: Winnipeg, MB Canada - 2015-04-24 *)
    M_QUANTUM_FUEL_SYSTEMS_TECHNOLOGIES_WORLDWIDE : UINT := 669; (* Manufacturer: Quantum Fuel Systems Technologies Worldwide, Inc | Location: Lake Forest, CA USA - *)
    M_STEMCO_LP : UINT := 670; (* Manufacturer: STEMCO LP | Location: Longview, TX USA - 2015-05-01 *)
    M_INNOVATIVE_CONTROLS : UINT := 671; (* Manufacturer: Innovative Controls Inc. | Location: East Pittsburgh, PA USA - 2015-05-05 *)
    M_OPTIMA_CONCEPT : UINT := 672; (* Manufacturer: OPTIMA Concept | Location: Ruitz, France - 2015-05-19 *)
    M_CARUELLE_NICOLAS : UINT := 673; (* Manufacturer: Caruelle Nicolas | Location: Saint Denis de l'Hotel, France - 2015-05-28 *)
    M_YARA_INTERNATIONAL_ASA : UINT := 674; (* Manufacturer: Yara International ASA | Location: Oslo, Norway - 2015-05-28 *)
    M_KAWASAKI_MOTORS : UINT := 675; (* Manufacturer: Kawasaki Motors, Ltd. (formerly Kawasaki Motors Corp., USA) | Location: Akashi, *)
    M_DANFOSS_IXA : UINT := 676; (* Manufacturer: Danfoss IXA A/S | Location: Vejle, Denmark - 2015-06-22 *)
    M_DSA_DATEN_UND_SYSTEMTECHNIK : UINT := 677; (* Manufacturer: DSA Daten- und Systemtechnik GmbH | Location: Aachen, Germany - 2015-06-29 *)
    M_KEEPTRUCKIN : UINT := 678; (* Manufacturer: KeepTruckin, Inc. | Location: Amherst, NY USA - 2015-06-30 *)
    M_OXE_MARINE : UINT := 679; (* Manufacturer: OXE Marine AB (formerly Cimco Marine AB) | Location: Ängelholm, Sweden - 2020-03-03 *)
    M_AMVAC_CHEMICAL : UINT := 680; (* Manufacturer: AMVAC Chemical Corporation | Location: Newport Beach, CA USA - 2015-07-14 *)
    M_BEDIA_MOTORENTECHNIK_AND : UINT := 681; (* Manufacturer: BEDIA Motorentechnik GmbH & Co. KG | Location: Altdorf bei Nuernberg, Germany - *)
    M_ECKELMANN_AG : UINT := 682; (* Manufacturer: Eckelmann AG | Location: Wiesbaden, Germany - 2015-07-27 *)
    M_FOSEN_ELEKTRO : UINT := 683; (* Manufacturer: Fosen Elektro | Location: Hasselvika, Norway - 2015-07-27 *)
    M_KEB : UINT := 684; (* Manufacturer: KEB | Location: Barntrup, Germany - 2015-07-27 *)
    M_ANEDO : UINT := 685; (* Manufacturer: ANEDO (formerly ANEDO Ltd.) | Location: Eydelstedt, Germany - 2019-05-24 *)
    M_TAIGENE_ELECTRIC_MACHINERY : UINT := 686; (* Manufacturer: Taigene Electric Machinery Corp. | Location: Taipei, Taiwan - 2015-07-27 *)
    M_FLIGHT_SYSTEMS : UINT := 687; (* Manufacturer: Flight Systems, Inc. | Location: Mechanicsburg, PA USA - 2015-07-31 *)
    M_ROCKFORD : UINT := 688; (* Manufacturer: Rockford Corp | Location: Tempe, AZ USA - 2015-07-31 *)
    M_AARCOMM_SYSTEMS : UINT := 689; (* Manufacturer: Aarcomm Systems Inc | Location: Coquitlam, BC Canada - 2015-07-31 *)
    M_LINAK : UINT := 690; (* Manufacturer: LINAK A/S | Location: Guderup, Denmark - 2015-08-03 *)
    M_DIGITROLL_AGRICULTURAL_ELECTRONICS : UINT := 691; (* Manufacturer: Digitroll Agricultural Electronics | Location: Hajduszoboszlo, Hungary - 2015-08-06 *)
    M_TANHAY : UINT := 692; (* Manufacturer: Tanhay Corporation | Location: Incheon, South Korea - 2015-08-13 *)
    M_AGILITY_FUEL_SOLUTIONS : UINT := 693; (* Manufacturer: Agility Fuel Solutions (formerly Agility Fuel Systems) | Location: Santa Ana, CA *)
    M_GASTOPS : UINT := 694; (* Manufacturer: GasTOPS Ltd. | Location: Ottawa, ON Canada - 2015-09-03 *)
    M_WELDON_TECHNOLOGIES : UINT := 695; (* Manufacturer: Weldon Technologies | Location: Columbus, OH USA - 2015-09-03 *)
    M_DRS_NETWORK_AND_IMAGING_SYSTEMS : UINT := 696; (* Manufacturer: DRS Network & Imaging Systems, LLC (DRS Technologies) | Location: Huntsville, AL *)
    M_JOST_UME : UINT := 697; (* Manufacturer: JOST Umeå AB (formerly Ålö AB) | Location: Umeå, Sweden - 2025-12-08 *)
    M_SCORPION_TECHNOLOGIES : UINT := 698; (* Manufacturer: Scorpion Technologies Ltd. | Location: Kamloops, BC Canada - 2015-10-13 *)
    M_HARMAN_INTERNATIONAL : UINT := 699; (* Manufacturer: Harman International (formerly Harman International Industries) | Location: *)
    M_K_TEC_EARTHMOVERS : UINT := 700; (* Manufacturer: K-Tec Earthmovers Inc. | Location: Rosenort, MB Canada - 2015-10-13 *)
    M_BIGROAD : UINT := 701; (* Manufacturer: BigRoad Inc. | Location: Kitchener, ON Canada - 2015-10-13 *)
    M_WEICHAI_POWER : UINT := 702; (* Manufacturer: Weichai Power Co., Ltd. | Location: Weifang, China - 2015-10-13 *)
    M_HYDRO_TAB_MARINE_ENGINEERING : UINT := 703; (* Manufacturer: Hydro Tab Marine Engineering | Location: Athens, Greece - 2015-10-13 *)
    M_JL_AUDIO : UINT := 704; (* Manufacturer: JL Audio, Inc. | Location: Miramar, FL USA - 2015-10-15 *)
    M_SVAB_HYDRAULIK : UINT := 705; (* Manufacturer: SVAB Hydraulik AB | Location: Hallsberg, Sweden - 2015-10-18 *)
    M_SHANGHAI_DIESEL_ENGINE_LIMITED : UINT := 706; (* Manufacturer: Shanghai Diesel Engine Corporation Limited | Location: Shanghai, China - 2015-10-22 *)
    M_ROCHESTER_GAUGES : UINT := 707; (* Manufacturer: Rochester Gauges Inc | Location: Dallas, TX USA - 2015-10-26 *)
    M_LARS_THRANE : UINT := 708; (* Manufacturer: Lars Thrane A/S | Location: Vedbaek, Denmark - 2015-10-26 *)
    M_MARQUARDT : UINT := 709; (* Manufacturer: Marquardt GmbH | Location: Rietheim-Weilheim, Germany - 2015-10-29 *)
    M_GREENTRONICS : UINT := 710; (* Manufacturer: Greentronics Ltd. | Location: Elmira, ON Canada - 2015-11-23 *)
    M_DAS : UINT := 711; (* Manufacturer: DAS Co., LTD | Location: Hwaseong-si, South Korea - 2015-11-23 *)
    M_LOR_MANUFACTURING_COMPANY : UINT := 712; (* Manufacturer: LOR Manufacturing Company Inc. | Location: Weidman, MI USA - 2015-11-23 *)
    M_US_HYBRID : UINT := 713; (* Manufacturer: US Hybrid Corporation | Location: Torrance, CA USA - 2015-12-09 *)
    M_KOBASHI_KOGYO : UINT := 714; (* Manufacturer: Kobashi Kogyo Co., Ltd. | Location: Okayama, Japan - 2015-12-09 *)
    M_AUTONNIC_RESEARCH : UINT := 715; (* Manufacturer: Autonnic Research Ltd | Location: Tollesbury, Essex UK - 2015-12-09 *)
    M_EATON_CONTROL_AND_POWER_CONVERSION_DIVISION : UINT := 716; (* Manufacturer: Eaton Control & Power Conversion Division (CPCD) | Location: Tualatin, OR USA - *)
    M_YACHT_DEVICES : UINT := 717; (* Manufacturer: Yacht Devices Ltd | Location: Kaliningrad, Russia - 2015-12-28 *)
    M_MICRONET : UINT := 718; (* Manufacturer: Micronet Inc | Location: Salt Lake City, UT USA - 2016-01-05 *)
    M_COJALI_S_L : UINT := 719; (* Manufacturer: Cojali S. L. | Location: Campo de Criptana, Spain - 2016-01-10 *)
    M_WITZ : UINT := 720; (* Manufacturer: WITZ Corporation | Location: Nagoya City, Japan - 2016-01-11 *)
    M_HYPRO : UINT := 721; (* Manufacturer: Hypro | Location: New Brighton, MN USA - 2016-01-13 *)
    M_CONTELEC_AG : UINT := 722; (* Manufacturer: Contelec AG | Location: Biel/Bienne, Switzerland - 2016-01-21 *)
    M_JABIL : UINT := 723; (* Manufacturer: Jabil Inc. | Location: Auburn Hills, MI USA - 2016-01-22 *)
    M_ELECTRONIC_APPLICATIONS : UINT := 724; (* Manufacturer: Electronic Applications, Inc. | Location: Phoenix, AZ USA - 2016-01-26 *)
    M_HITACHI_CONSTRUCTION_MACHINERY : UINT := 725; (* Manufacturer: Hitachi Construction Machinery Co., Ltd. | Location: Kandatsu-machi, Japan - *)
    M_MIDORI_PRECISIONS : UINT := 726; (* Manufacturer: MIDORI PRECISIONS | Location: Tokyo, Japan - 2016-02-03 *)
    M_DHOOT_TRANSMISSION_PVT : UINT := 727; (* Manufacturer: Dhoot Transmission Pvt Ltd. | Location: Aurangabad, India - 2016-02-18 *)
    M_STREUMASTER : UINT := 728; (* Manufacturer: Streumaster (formerly Streumaster / Panien) | Location: Egglkofen, Germany - *)
    M_LIEBHERR : UINT := 729; (* Manufacturer: Liebherr | Location: Bulle, Switzerland - 2016-03-02 *)
    M_BERTHOUD_AGRICOLE : UINT := 730; (* Manufacturer: BERTHOUD AGRICOLE | Location: Belleville sur Saone, France - 2016-03-03 *)
    M_MODINE_MANUFACTURING_COMPANY : UINT := 731; (* Manufacturer: Modine Manufacturing Company | Location: Racine, WI USA - 2016-03-04 *)
    M_GEFRAN : UINT := 732; (* Manufacturer: Gefran S.p.A. | Location: Provaglio d'Iseo, Italy - 2016-03-04 *)
    M_INTENDIA_S_L : UINT := 733; (* Manufacturer: Intendia S.L. | Location: Madrid, Spain - 2016-03-23 *)
    M_REAPSYSTEMS : UINT := 734; (* Manufacturer: REAPsystems | Location: St Denys, Southampton UK - 2016-03-23 *)
    M_AEM_PERFORMANCE_ELECTRONICS : UINT := 735; (* Manufacturer: AEM Performance Electronics | Location: Hawthorne, CA USA - 2016-03-23 *)
    M_TEREX_AERIAL_WORK_PLATFORMS_GENIE : UINT := 736; (* Manufacturer: Terex Aerial Work Platforms - Genie | Location: Redmond, WA USA - 2016-04-21 *)
    M_BALLUFF : UINT := 737; (* Manufacturer: Balluff GmbH | Location: Neuhausen, Germany - 2016-04-29 *)
    M_BLUE_INK_TECHNOLOGIES : UINT := 738; (* Manufacturer: Blue Ink Technologies | Location: Huntington, WV USA - 2016-05-04 *)
    M_LXNAV_D_O_O : UINT := 739; (* Manufacturer: LXNAV d.o.o. | Location: Celje, Slovenia - 2016-05-19 *)
    M_E_TRACTION : UINT := 740; (* Manufacturer: e-Traction | Location: Apeldoorn, The Netherlands - 2016-05-19 *)
    M_CARLING_TECHNOLOGIES : UINT := 741; (* Manufacturer: Carling Technologies | Location: Plainville, CT USA - 2016-05-19 *)
    M_EROAD : UINT := 742; (* Manufacturer: EROAD | Location: Auckland, New Zealand - 2016-05-22 *)
    M_DAEMYUNG_ELEVATOR : UINT := 743; (* Manufacturer: Daemyung Elevator Co., Ltd. | Location: Ulsan, Republic of Korea - 2016-05-25 *)
    M_WOOSUNG_ENGINEERING : UINT := 744; (* Manufacturer: Woosung Engineering Co., Ltd. | Location: Gyengsangnam-do, Republic of Korea - *)
    M_CIDRA_CORPORATE_SERVICES : UINT := 745; (* Manufacturer: Cidra Corporate Services Inc. | Location: Wallingford, CT USA - 2016-06-10 *)
    M_SUREPOINT_AG_SYSTEMS : UINT := 746; (* Manufacturer: SurePoint Ag Systems (formerly SureFire Ag Systems, Inc.) | Location: Atwood, KS *)
    M_AGRATRONIX : UINT := 747; (* Manufacturer: Agratronix | Location: Streetsboro, OH USA - 2016-06-10 *)
    M_ISOTTA : UINT := 748; (* Manufacturer: ISOTTA | Location: Occhiobello, Italy - 2016-06-10 *)
    M_CHART : UINT := 749; (* Manufacturer: Chart Inc. | Location: Ball Ground, GA USA - 2016-06-20 *)
    M_JOSKIN : UINT := 750; (* Manufacturer: Joskin SA | Location: Soumagne, Belgium - 2016-06-20 *)
    M_PACIFIC_TRACK : UINT := 751; (* Manufacturer: Pacific Track | Location: Newport Beach, CA USA - 2016-06-24 *)
    M_DEEP_SEA_ELECTRONICS_PLC : UINT := 752; (* Manufacturer: Deep Sea Electronics Plc | Location: Hunmanby, North Yorkshire UK - 2016-06-24 *)
    M_AIROD_TECHNOLOGIES : UINT := 753; (* Manufacturer: AIROD Technologies | Location: Toulouse, France - 2016-06-29 *)
    M_PARKER_HANNIFIN_AUTOMATION_GROUP : UINT := 754; (* Manufacturer: Parker Hannifin Corp., Automation Group | Location: Cleveland, OH USA - 2016-07-01 *)
    M_FIREFLY_INTEGRATIONS : UINT := 755; (* Manufacturer: Firefly Integrations | Location: Middlebury, IN USA - 2016-07-21 *)
    M_MASCHIO_GASPARDO : UINT := 756; (* Manufacturer: Maschio Gaspardo S.P.A. | Location: Campodarsego, Italy - 2016-07-21 *)
    M_IMPCO_TECHNOLOGIES : UINT := 757; (* Manufacturer: IMPCO Technologies | Location: Calgary, AB Canada - 2016-07-21 *)
    M_BANNER_ENGINEERING : UINT := 758; (* Manufacturer: Banner Engineering Corp. | Location: Minneapolis, MN USA - 2016-07-21 *)
    M_HYDRO_GEAR : UINT := 759; (* Manufacturer: Hydro-Gear | Location: Sullivan, IL USA - 2016-07-28 *)
    M_BERNECKER_RAINER_INDUSTRIE_ELEKTRONIK : UINT := 760; (* Manufacturer: Bernecker + Rainer Industrie Elektronik GmbH | Location: Eggelsberg, Austria - *)
    M_MITA_OLEODINAMICA : UINT := 761; (* Manufacturer: MITA OLEODINAMICA S.p.A. | Location: Tregnago, Italy - 2016-07-28 *)
    M_ROJ_S_R_L : UINT := 762; (* Manufacturer: ROJ s.r.l. | Location: Biella, Italy - 2016-08-01 *)
    M_AT_SYSTEMS_BVBA : UINT := 763; (* Manufacturer: AT-Systems BVBA | Location: Meerle, Belgium - 2016-08-02 *)
    M_BEDNAR_FMT_S_R_O : UINT := 764; (* Manufacturer: Bednar FMT s.r.o. | Location: Prague, Czech Republic - 2016-08-17 *)
    M_GIGAVAC : UINT := 765; (* Manufacturer: GIGAVAC | Location: Carpinteria, CA USA - 2016-08-17 *)
    M_EPEC_OY : UINT := 766; (* Manufacturer: Epec Oy | Location: Seinajoki, Finland - 2016-08-17 *)
    M_ALLIANCE_WIRELESS_TECHNOLOGIES : UINT := 767; (* Manufacturer: Alliance Wireless Technologies Inc. | Location: Houston, TX USA - 2016-08-30 *)
    M_FLORES_AUTOMATION : UINT := 768; (* Manufacturer: Flores Automation, LLC | Location: Muskego, WI USA - 2016-08-30 *)
    M_TROMBETTA : UINT := 769; (* Manufacturer: Trombetta | Location: Milwaukee, WI USA - 2016-08-30 *)
    M_MONOSEM : UINT := 770; (* Manufacturer: MONOSEM | Location: Largeasse, France - 2016-08-30 *)
    M_SHAW_DEVELOPMENT : UINT := 771; (* Manufacturer: Shaw Development, LLC | Location: Bonita Springs, FL USA - 2016-09-12 *)
    M_BLINK_MARINE : UINT := 772; (* Manufacturer: Blink Marine | Location: Milano, Italy - 2016-09-30 *)
    M_CLARION_OF_AMERICA : UINT := 773; (* Manufacturer: Clarion Corporation of America | Location: Cypress, CA USA - 2016-09-30 *)
    M_TAISHO : UINT := 774; (* Manufacturer: Taisho Corporation | Location: Mito, Japan - 2016-09-30 *)
    M_ZIEHL_ABEGG_AUTOMOTIVE : UINT := 775; (* Manufacturer: ZIEHL-ABEGG Automotive GmbH | Location: Kupferzell, Germany - 2016-10-14 *)
    M_HMI_SYSTEMS : UINT := 776; (* Manufacturer: HMI Systems LLC | Location: Lakeland, FL USA - 2016-10-25 *)
    M_OCEAN_SIGNAL : UINT := 777; (* Manufacturer: Ocean Signal Ltd | Location: Margate, Kent UK - 2016-10-25 *)
    M_SEAKEEPER : UINT := 778; (* Manufacturer: Seakeeper Inc. | Location: California, MD USA - 2016-10-25 *)
    M_RLC_ELECTRONIC_SYSTEMS : UINT := 779; (* Manufacturer: RLC Electronic Systems | Location: Sinking Spring, PA USA - 2016-11-01 *)
    M_TURNTIDE_TRANSPORT_LIMITED : UINT := 780; (* Manufacturer: Turntide Transport Limited (formerly AVID Technology Ltd) | Location: Cramlington, *)
    M_POLY_PLANAR : UINT := 781; (* Manufacturer: Poly-Planar LLC | Location: Hanover, MD USA - 2016-11-04 *)
    M_AVR_NV : UINT := 782; (* Manufacturer: AVR nv | Location: Roeselare, Belgium - 2019-12-14 *)
    M_LOUP_ELECTRONICS : UINT := 783; (* Manufacturer: Loup Electronics Inc. | Location: Lincoln, NE USA - 2016-12-02 *)
    M_CM_AUTOMOTIVE_SYSTEMS : UINT := 784; (* Manufacturer: CM Automotive Systems, Inc. | Location: Walnut, CA USA - 2016-12-02 *)
    M_FISCHER_PANDA : UINT := 785; (* Manufacturer: Fischer Panda GmbH | Location: Paderborn, Germany - 2016-12-17 *)
    M_JOHNSON_MATTHEY_BATTERY_SYSTEMS : UINT := 786; (* Manufacturer: Johnson Matthey Battery Systems | Location: Milton Keynes, Bucks UK - 2016-12-17 *)
    M_ABERTAX_TECHNOLOGIES_LIMITED : UINT := 787; (* Manufacturer: Abertax Technologies Limited | Location: Paola, Malta - 2017-01-15 *)
    M_MOTEC_PTY : UINT := 788; (* Manufacturer: MoTeC Pty Ltd | Location: Melbourne, Victoria Australia - 2017-01-15 *)
    M_GRADALL : UINT := 789; (* Manufacturer: GRADALL | Location: New Philadelphia, OH USA - 2017-02-03 *)
    M_VACALL : UINT := 790; (* Manufacturer: VACALL | Location: New Philadelphia, OH USA - 2017-02-03 *)
    M_AUTEC : UINT := 791; (* Manufacturer: AUTEC | Location: Caldogno, Italy - 2017-02-07 *)
    M_KOSTAL_MEXICANA : UINT := 792; (* Manufacturer: Kostal Mexicana | Location: Querétaro, Mexico - 2017-02-07 *)
    M_JAMES_FISHER_PROLEC : UINT := 793; (* Manufacturer: James Fisher Prolec | Location: Poole, Dorset UK - 2017-02-09 *)
    M_SHIHLIN_ELECTRIC_AND_ENGINEERING : UINT := 794; (* Manufacturer: Shihlin Electric & Engineering Corporation | Location: Suzhou, China - 2017-02-09 *)
    M_BROYDA_ENTERPRISES_PTY : UINT := 795; (* Manufacturer: Broyda Enterprises Pty Ltd | Location: Sydney, Australia - 2017-02-10 *)
    M_CANADIAN_AUTOMOTIVE_INDUSTRIES : UINT := 796; (* Manufacturer: Canadian Automotive Industries Ltd | Location: Stony Plain, AB Canada - 2017-02-10 *)
    M_TIDES_MARINE : UINT := 797; (* Manufacturer: Tides Marine | Location: Deerfield Beach, FL USA - 2017-02-10 *)
    M_LUMISHORE : UINT := 798; (* Manufacturer: Lumishore Ltd | Location: Swansea, Wales UK - 2017-02-10 *)
    M_STILLWATER_DESIGNS_AND_AUDIO_KICKER : UINT := 799; (* Manufacturer: Stillwater Designs and Audio, Inc. - KICKER | Location: Stillwater, OK USA - *)
    M_DELTA_Q_TECHNOLOGIES : UINT := 800; (* Manufacturer: Delta-Q Technologies | Location: Burnaby, BC Canada - 2017-02-16 *)
    M_LOR_MANUFACTURING_COMPANY_801 : UINT := 801; (* Manufacturer: LOR Manufacturing Company Inc. | Location: Weidman, MI USA - 2017-03-01 *)
    M_SPBI : UINT := 802; (* Manufacturer: SPBI (Bj Technologie) | Location: Dompierre-sur-Yon, France - 2017-03-01 *)
    M_GILL_SENSORS_AND_CONTROLS_LIMITED : UINT := 803; (* Manufacturer: Gill Sensors & Controls Limited | Location: Lymington, Hampshire UK - 2017-03-03 *)
    M_ASA_ELECTRONICS : UINT := 804; (* Manufacturer: ASA Electronics | Location: Elkhart, IN USA - 2017-03-09 *)
    M_GUNDERSEN_AND_L_KEN : UINT := 805; (* Manufacturer: Gundersen & Løken AS | Location: Oslo, Norway - 2017-03-17 *)
    M_CHARGE_AUTOMOTIVE : UINT := 806; (* Manufacturer: Charge Automotive Ltd | Location: Banbury, Oxfordshire UK - 2017-03-17 *)
    M_SCHNEIDER_ELECTRIC : UINT := 807; (* Manufacturer: Schneider-Electric | Location: Burnaby, BC Canada - 2017-03-27 *)
    M_RIMEX_SUPPLY : UINT := 808; (* Manufacturer: RIMEX Supply Ltd. | Location: Surrey, BC Canada - 2017-03-27 *)
    M_HMS_INDUSTRIAL_NETWORKS : UINT := 809; (* Manufacturer: HMS Industrial Networks AB | Location: Halmstad, Sweden - 2017-04-04 *)
    M_DUTCH_POWER_COMPANY : UINT := 810; (* Manufacturer: Dutch Power Company | Location: Giessen, The Netherlands - 2017-04-07 *)
    M_BLUE_WATER_DESALINATION : UINT := 811; (* Manufacturer: Blue Water Desalination | Location: Carson, CA USA - 2017-04-10 *)
    M_TORCH_TECHNOLOGIES : UINT := 812; (* Manufacturer: Torch Technologies | Location: Huntsville, AL USA - 2017-04-12 *)
    M_THALES_SUISSE : UINT := 813; (* Manufacturer: Thales Suisse SA | Location: Zurich, Switzerland - 2017-04-12 *)
